ABB RAPID module: ReplayTargets_v20.mod

MODULE ReplayTargets_v20
    ! Generated from tests_v20.csv and success_v20.csv.
    ! Target names include version and testId. B* variants include version, testId, and confId.

    ! Robtargets and jointtargets for replay
    CONST robtarget rA_v20_t1 := [[2348.43,-0.0291239,345.047],[0.199058,0.678508,0.678515,0.199049],[-1,-1,-4,0],[9E+09,9E+09,9E+09,9E+09,9E+09,9E+09]];
    CONST robtarget rB_v20_t1 := [[2448.23,15.5994,307.458],[0.265046,0.716851,0.60792,0.215193],[-1,-1,-4,0],[9E+09,9E+09,9E+09,9E+09,9E+09,9E+09]];
    CONST robtarget rB_v20_t1_c2 := [[2448.23,15.5994,307.458],[0.265046,0.716851,0.60792,0.215193],[0,0,-4,0],[9E+09,9E+09,9E+09,9E+09,9E+09,9E+09]];
    CONST jointtarget jA_v20_t1 := [[-0.000703123,42.2,5.7,-0.000639588,9.4,-270.001],[9E+09,9E+09,9E+09,9E+09,9E+09,9E+09]];
    CONST jointtarget jB_v20_t1 := [[44.9994,-58.7,29.3,-90.0002,39.2,-360.001],[9E+09,9E+09,9E+09,9E+09,9E+09,9E+09]];
    CONST jointtarget jBseed_v20_t1 := [[0,42.2,5.7,0,9.4,-270],[9E+09,9E+09,9E+09,9E+09,9E+09,9E+09]];
    CONST num seedB_v20_t1 := 26880;

    CONST robtarget rA_v20_t2 := [[-1479.72,1306.42,1538.84],[0.318675,0.68714,-0.344424,-0.554668],[1,-4,-1,0],[9E+09,9E+09,9E+09,9E+09,9E+09,9E+09]];
    CONST robtarget rB_v20_t2 := [[-1474.64,1359.47,1499.34],[0.343208,0.716755,-0.240423,-0.557376],[1,-4,-1,0],[9E+09,9E+09,9E+09,9E+09,9E+09,9E+09]];
    CONST robtarget rB_v20_t2_c4 := [[-1474.64,1359.47,1499.34],[0.343208,0.716755,-0.240423,-0.557376],[0,-4,0,0],[9E+09,9E+09,9E+09,9E+09,9E+09,9E+09]];
    CONST jointtarget jA_v20_t2 := [[135,-0.2,15.7,-270,47.2,-45.0005],[9E+09,9E+09,9E+09,9E+09,9E+09,9E+09]];
    CONST jointtarget jB_v20_t2 := [[44.9994,-58.7,29.3,-90.0002,39.2,-360.001],[9E+09,9E+09,9E+09,9E+09,9E+09,9E+09]];
    CONST jointtarget jBseed_v20_t2 := [[135,-0.2,15.7,-270,47.2,-45],[9E+09,9E+09,9E+09,9E+09,9E+09,9E+09]];
    CONST num seedB_v20_t2 := 8986;

    CONST robtarget rA_v20_t3 := [[-971.424,971.394,2079.64],[1.34054E-5,0.567678,-0.567677,-0.596225],[1,0,-4,0],[9E+09,9E+09,9E+09,9E+09,9E+09,9E+09]];
    CONST robtarget rB_v20_t3 := [[-1027.84,1052.99,2102.83],[0.00324872,0.494172,-0.597172,-0.631798],[1,0,-4,0],[9E+09,9E+09,9E+09,9E+09,9E+09,9E+09]];
    CONST robtarget rB_v20_t3_c2 := [[-1027.84,1052.99,2102.83],[0.00324872,0.494172,-0.597172,-0.631798],[0,0,-4,0],[9E+09,9E+09,9E+09,9E+09,9E+09,9E+09]];
    CONST jointtarget jA_v20_t3 := [[135.001,-31.4,20,0.000962912,28.2,-315],[9E+09,9E+09,9E+09,9E+09,9E+09,9E+09]];
    CONST jointtarget jB_v20_t3 := [[44.9994,-58.7,29.3,-90.0002,39.2,-360.001],[9E+09,9E+09,9E+09,9E+09,9E+09,9E+09]];
    CONST jointtarget jBseed_v20_t3 := [[135,-31.4,20,0,28.2,-315],[9E+09,9E+09,9E+09,9E+09,9E+09,9E+09]];
    CONST num seedB_v20_t3 := 10305;

    CONST robtarget rA_v20_t4 := [[-87.9993,-1983.55,1057.37],[0.0429391,-0.444605,-0.7263,0.522466],[-1,2,-4,0],[9E+09,9E+09,9E+09,9E+09,9E+09,9E+09]];
    CONST robtarget rB_v20_t4 := [[-13.7229,-1932.17,1079.47],[0.049502,-0.443461,-0.708683,0.546499],[-1,2,-4,0],[9E+09,9E+09,9E+09,9E+09,9E+09,9E+09]];
    CONST robtarget rB_v20_t4_c3 := [[-13.7229,-1932.17,1079.47],[0.049502,-0.443461,-0.708683,0.546499],[0,4,-4,0],[9E+09,9E+09,9E+09,9E+09,9E+09,9E+09]];
    CONST jointtarget jA_v20_t4 := [[-89.9999,6.4,25.6,270,31.8,-315],[9E+09,9E+09,9E+09,9E+09,9E+09,9E+09]];
    CONST jointtarget jB_v20_t4 := [[44.9994,-58.7,29.3,-90.0002,39.2,-360.001],[9E+09,9E+09,9E+09,9E+09,9E+09,9E+09]];
    CONST jointtarget jBseed_v20_t4 := [[-90,6.4,25.6,270,31.8,-315],[9E+09,9E+09,9E+09,9E+09,9E+09,9E+09]];
    CONST num seedB_v20_t4 := 13879;

    CONST robtarget rA_v20_t5 := [[-1618.75,1500.97,2623.16],[0.821125,-0.204966,-0.515033,0.135956],[1,1,1,0],[9E+09,9E+09,9E+09,9E+09,9E+09,9E+09]];
    CONST robtarget rB_v20_t5 := [[-1548.36,1545.2,2531.64],[0.862384,-0.207508,-0.444636,0.124636],[1,1,1,0],[9E+09,9E+09,9E+09,9E+09,9E+09,9E+09]];
    CONST robtarget rB_v20_t5_c5 := [[-1548.36,1545.2,2531.64],[0.862384,-0.207508,-0.444636,0.124636],[0,0,0,0],[9E+09,9E+09,9E+09,9E+09,9E+09,9E+09]];
    CONST jointtarget jA_v20_t5 := [[135.001,24.2,-50.6,90.0008,29.9,135],[9E+09,9E+09,9E+09,9E+09,9E+09,9E+09]];
    CONST jointtarget jB_v20_t5 := [[44.9994,-58.7,29.3,-90.0002,39.2,-360.001],[9E+09,9E+09,9E+09,9E+09,9E+09,9E+09]];
    CONST jointtarget jBseed_v20_t5 := [[135,24.2,-50.6,90,29.9,135],[9E+09,9E+09,9E+09,9E+09,9E+09,9E+09]];
    CONST num seedB_v20_t5 := 13200;

    CONST robtarget rA_v20_t6 := [[-0.00301178,-325.583,2816.94],[0.976672,0.214735,1.31208E-6,-1.04287E-5],[-2,-3,-2,0],[9E+09,9E+09,9E+09,9E+09,9E+09,9E+09]];
    CONST robtarget rB_v20_t6 := [[12.1082,-256.874,2819],[0.966244,0.241594,-0.061799,0.0646911],[-2,-3,-2,0],[9E+09,9E+09,9E+09,9E+09,9E+09,9E+09]];
    CONST robtarget rB_v20_t6_c4 := [[12.1082,-256.874,2819],[0.966244,0.241594,-0.061799,0.0646911],[0,-4,0,0],[9E+09,9E+09,9E+09,9E+09,9E+09,9E+09]];
    CONST jointtarget jA_v20_t6 := [[-90.0006,-53,2.5,-180.001,14.7,-90.0001],[9E+09,9E+09,9E+09,9E+09,9E+09,9E+09]];
    CONST jointtarget jB_v20_t6 := [[44.9994,-58.7,29.3,-90.0002,39.2,-360.001],[9E+09,9E+09,9E+09,9E+09,9E+09,9E+09]];
    CONST jointtarget jBseed_v20_t6 := [[-90,-53,2.5,-180,14.7,-90],[9E+09,9E+09,9E+09,9E+09,9E+09,9E+09]];
    CONST num seedB_v20_t6 := 26677;

    CONST robtarget rA_v20_t7 := [[1448.08,-93.8143,1159.42],[0.151545,0.78397,-0.512149,0.316431],[-1,-1,-2,0],[9E+09,9E+09,9E+09,9E+09,9E+09,9E+09]];
    CONST robtarget rB_v20_t7 := [[1454.33,-138.013,1185.15],[0.132933,0.822904,-0.460863,0.304569],[-1,-1,-2,0],[9E+09,9E+09,9E+09,9E+09,9E+09,9E+09]];
    CONST robtarget rB_v20_t7_c5 := [[1454.33,-138.013,1185.15],[0.132933,0.822904,-0.460863,0.304569],[0,0,0,0],[9E+09,9E+09,9E+09,9E+09,9E+09,9E+09]];
    CONST robtarget rB_v20_t7_c8 := [[1454.33,-138.013,1185.15],[0.132933,0.822904,-0.460863,0.304569],[0,0,4,0],[9E+09,9E+09,9E+09,9E+09,9E+09,9E+09]];
    CONST jointtarget jA_v20_t7 := [[-0.000199191,-22.7,45.6,-44.9996,52.6,-90.0001],[9E+09,9E+09,9E+09,9E+09,9E+09,9E+09]];
    CONST jointtarget jB_v20_t7 := [[44.9994,-58.7,29.3,-90.0002,39.2,-360.001],[9E+09,9E+09,9E+09,9E+09,9E+09,9E+09]];
    CONST jointtarget jBseed_v20_t7 := [[0,-22.7,45.6,-45,52.6,-90],[9E+09,9E+09,9E+09,9E+09,9E+09,9E+09]];
    CONST num seedB_v20_t7 := 27772;

    CONST robtarget rA_v20_t8 := [[1676.32,-1692.34,1208.08],[0.539776,0.76394,0.296429,0.192788],[-1,2,2,0],[9E+09,9E+09,9E+09,9E+09,9E+09,9E+09]];
    CONST robtarget rB_v20_t8 := [[1594.8,-1750.16,1141.03],[0.532215,0.796727,0.236675,0.161115],[-1,2,2,0],[9E+09,9E+09,9E+09,9E+09,9E+09,9E+09]];
    CONST robtarget rB_v20_t8_c5 := [[1594.8,-1750.16,1141.03],[0.532215,0.796727,0.236675,0.161115],[0,0,0,0],[9E+09,9E+09,9E+09,9E+09,9E+09,9E+09]];
    CONST robtarget rB_v20_t8_c6 := [[1594.8,-1750.16,1141.03],[0.532215,0.796727,0.236675,0.161115],[0,4,0,0],[9E+09,9E+09,9E+09,9E+09,9E+09,9E+09]];
    CONST jointtarget jA_v20_t8 := [[-45.0002,21.5,2.5,225,5.5,225.001],[9E+09,9E+09,9E+09,9E+09,9E+09,9E+09]];
    CONST jointtarget jB_v20_t8 := [[44.9994,-58.7,29.3,-90.0002,39.2,-360.001],[9E+09,9E+09,9E+09,9E+09,9E+09,9E+09]];
    CONST jointtarget jBseed_v20_t8 := [[-45,21.5,2.5,225,5.5,225],[9E+09,9E+09,9E+09,9E+09,9E+09,9E+09]];
    CONST num seedB_v20_t8 := 3525;

    CONST robtarget rA_v20_t9 := [[-1079.34,1079.34,1641.75],[0.71135,-0.589521,-0.244195,0.294643],[1,1,0,0],[9E+09,9E+09,9E+09,9E+09,9E+09,9E+09]];
    CONST robtarget rB_v20_t9 := [[-966.677,1102.66,1605.56],[0.710962,-0.602204,-0.160651,0.325692],[1,1,0,0],[9E+09,9E+09,9E+09,9E+09,9E+09,9E+09]];
    CONST robtarget rB_v20_t9_c4 := [[-966.677,1102.66,1605.56],[0.710962,-0.602204,-0.160651,0.325692],[0,-4,0,0],[9E+09,9E+09,9E+09,9E+09,9E+09,9E+09]];
    CONST robtarget rB_v20_t9_c5 := [[-966.677,1102.66,1605.56],[0.710962,-0.602204,-0.160651,0.325692],[0,0,0,0],[9E+09,9E+09,9E+09,9E+09,9E+09,9E+09]];
    CONST jointtarget jA_v20_t9 := [[135,-27.5,36.8,179.999,20,89.9998],[9E+09,9E+09,9E+09,9E+09,9E+09,9E+09]];
    CONST jointtarget jB_v20_t9 := [[44.9994,-58.7,29.3,-90.0002,39.2,-360.001],[9E+09,9E+09,9E+09,9E+09,9E+09,9E+09]];
    CONST jointtarget jBseed_v20_t9 := [[135,-27.5,36.8,180,20,90],[9E+09,9E+09,9E+09,9E+09,9E+09,9E+09]];
    CONST num seedB_v20_t9 := 19894;

    CONST robtarget rA_v20_t10 := [[138.442,2028.98,2186.31],[0.730348,-0.405331,0.548774,-0.0338534],[1,-1,-4,0],[9E+09,9E+09,9E+09,9E+09,9E+09,9E+09]];
    CONST robtarget rB_v20_t10 := [[136.362,1909.01,2210.89],[0.67858,-0.463529,0.560222,-0.104029],[1,-1,-4,0],[9E+09,9E+09,9E+09,9E+09,9E+09,9E+09]];
    CONST robtarget rB_v20_t10_c2 := [[136.362,1909.01,2210.89],[0.67858,-0.463529,0.560222,-0.104029],[0,0,-4,0],[9E+09,9E+09,9E+09,9E+09,9E+09,9E+09]];
    CONST jointtarget jA_v20_t10 := [[90.0002,5.4,-12.5,-89.9994,56,-315],[9E+09,9E+09,9E+09,9E+09,9E+09,9E+09]];
    CONST jointtarget jB_v20_t10 := [[44.9994,-58.7,29.3,-90.0002,39.2,-360.001],[9E+09,9E+09,9E+09,9E+09,9E+09,9E+09]];
    CONST jointtarget jBseed_v20_t10 := [[90,5.4,-12.5,-90,56,-315],[9E+09,9E+09,9E+09,9E+09,9E+09,9E+09]];
    CONST num seedB_v20_t10 := 2946;

    CONST robtarget rA_v20_t11 := [[1156.13,1172.74,2229.26],[0.716045,-0.261719,0.561783,0.321221],[0,1,2,0],[9E+09,9E+09,9E+09,9E+09,9E+09,9E+09]];
    CONST robtarget rB_v20_t11 := [[1235.48,1131.05,2183.34],[0.723682,-0.214068,0.602425,0.259892],[0,1,2,0],[9E+09,9E+09,9E+09,9E+09,9E+09,9E+09]];
    CONST robtarget rB_v20_t11_c6 := [[1235.48,1131.05,2183.34],[0.723682,-0.214068,0.602425,0.259892],[0,4,0,0],[9E+09,9E+09,9E+09,9E+09,9E+09,9E+09]];
    CONST jointtarget jA_v20_t11 := [[45.0005,-17.1,7.7,135,5.7,225.001],[9E+09,9E+09,9E+09,9E+09,9E+09,9E+09]];
    CONST jointtarget jB_v20_t11 := [[44.9994,-58.7,29.3,-90.0002,39.2,-360.001],[9E+09,9E+09,9E+09,9E+09,9E+09,9E+09]];
    CONST jointtarget jBseed_v20_t11 := [[45,-17.1,7.7,135,5.7,225],[9E+09,9E+09,9E+09,9E+09,9E+09,9E+09]];
    CONST num seedB_v20_t11 := 2997;

    CONST robtarget rA_v20_t12 := [[2684.36,-73.5564,2199.23],[0.910091,0.192131,0.342612,-0.132052],[-1,-2,1,0],[9E+09,9E+09,9E+09,9E+09,9E+09,9E+09]];
    CONST robtarget rB_v20_t12 := [[2614.98,29.0324,2213.55],[0.904293,0.217033,0.287629,-0.228955],[-1,-2,1,0],[9E+09,9E+09,9E+09,9E+09,9E+09,9E+09]];
    CONST robtarget rB_v20_t12_c4 := [[2614.98,29.0324,2213.55],[0.904293,0.217033,0.287629,-0.228955],[0,-4,0,0],[9E+09,9E+09,9E+09,9E+09,9E+09,9E+09]];
    CONST jointtarget jA_v20_t12 := [[-0.000960234,53.1,-74.1,-135,38.5,135],[9E+09,9E+09,9E+09,9E+09,9E+09,9E+09]];
    CONST jointtarget jB_v20_t12 := [[44.9994,-58.7,29.3,-90.0002,39.2,-360.001],[9E+09,9E+09,9E+09,9E+09,9E+09,9E+09]];
    CONST jointtarget jBseed_v20_t12 := [[0,53.1,-74.1,-135,38.5,135],[9E+09,9E+09,9E+09,9E+09,9E+09,9E+09]];
    CONST num seedB_v20_t12 := 170;

    CONST robtarget rA_v20_t13 := [[0.00419857,298.28,3136.24],[0.368757,-0.102269,-0.246896,-0.890282],[0,-1,-3,0],[9E+09,9E+09,9E+09,9E+09,9E+09,9E+09]];
    CONST robtarget rB_v20_t13 := [[-28.1699,255.485,3048.95],[0.422465,-0.149707,-0.227149,-0.864589],[0,-1,-3,0],[9E+09,9E+09,9E+09,9E+09,9E+09,9E+09]];
    CONST robtarget rB_v20_t13_c5 := [[-28.1699,255.485,3048.95],[0.422465,-0.149707,-0.227149,-0.864589],[0,0,0,0],[9E+09,9E+09,9E+09,9E+09,9E+09,9E+09]];
    CONST jointtarget jA_v20_t13 := [[89.9992,-38.4,-22.1,-0.000207024,1.5,-225],[9E+09,9E+09,9E+09,9E+09,9E+09,9E+09]];
    CONST jointtarget jB_v20_t13 := [[44.9994,-58.7,29.3,-90.0002,39.2,-360.001],[9E+09,9E+09,9E+09,9E+09,9E+09,9E+09]];
    CONST jointtarget jBseed_v20_t13 := [[90,-38.4,-22.1,0,1.5,-225],[9E+09,9E+09,9E+09,9E+09,9E+09,9E+09]];
    CONST num seedB_v20_t13 := 21910;

    CONST robtarget rA_v20_t14 := [[-217.284,360.724,3378.8],[0.700643,0.169716,0.342315,0.602592],[1,2,-3,0],[9E+09,9E+09,9E+09,9E+09,9E+09,9E+09]];
    CONST robtarget rB_v20_t14 := [[-203.6,421.862,3270.5],[0.694668,0.134709,0.317582,0.631214],[1,2,-3,0],[9E+09,9E+09,9E+09,9E+09,9E+09,9E+09]];
    CONST robtarget rB_v20_t14_c3 := [[-203.6,421.862,3270.5],[0.694668,0.134709,0.317582,0.631214],[0,4,-4,0],[9E+09,9E+09,9E+09,9E+09,9E+09,9E+09]];
    CONST jointtarget jA_v20_t14 := [[135,-13.9,-53.2,224.999,59.2,-269.999],[9E+09,9E+09,9E+09,9E+09,9E+09,9E+09]];
    CONST jointtarget jB_v20_t14 := [[44.9994,-58.7,29.3,-90.0002,39.2,-360.001],[9E+09,9E+09,9E+09,9E+09,9E+09,9E+09]];
    CONST jointtarget jBseed_v20_t14 := [[135,-13.9,-53.2,225,59.2,-270],[9E+09,9E+09,9E+09,9E+09,9E+09,9E+09]];
    CONST num seedB_v20_t14 := 4792;

    CONST robtarget rA_v20_t15 := [[-1472.6,1608.71,1063.4],[0.00433901,0.101786,-0.642952,-0.7591],[1,2,2,0],[9E+09,9E+09,9E+09,9E+09,9E+09,9E+09]];
    CONST robtarget rB_v20_t15 := [[-1457.34,1584.84,1032.33],[0.104698,-0.085445,0.659952,0.739054],[1,2,2,0],[9E+09,9E+09,9E+09,9E+09,9E+09,9E+09]];
    CONST robtarget rB_v20_t15_c6 := [[-1457.34,1584.84,1032.33],[0.104698,-0.085445,0.659952,0.739054],[0,4,0,0],[9E+09,9E+09,9E+09,9E+09,9E+09,9E+09]];
    CONST jointtarget jA_v20_t15 := [[135,17.2,16.9,225.001,54.6,224.999],[9E+09,9E+09,9E+09,9E+09,9E+09,9E+09]];
    CONST jointtarget jB_v20_t15 := [[44.9994,-58.7,29.3,-90.0002,39.2,-360.001],[9E+09,9E+09,9E+09,9E+09,9E+09,9E+09]];
    CONST jointtarget jBseed_v20_t15 := [[135,17.2,16.9,225,54.6,225],[9E+09,9E+09,9E+09,9E+09,9E+09,9E+09]];
    CONST num seedB_v20_t15 := 4784;

    CONST robtarget rA_v20_t17 := [[-0.0178469,-1454.99,2120.23],[0.807655,0.448611,-0.185819,0.334533],[-2,-3,3,0],[9E+09,9E+09,9E+09,9E+09,9E+09,9E+09]];
    CONST robtarget rB_v20_t17 := [[95.0666,-1392.8,2093],[0.815027,0.420993,-0.246161,0.312891],[-2,-3,3,0],[9E+09,9E+09,9E+09,9E+09,9E+09,9E+09]];
    CONST robtarget rB_v20_t17_c7 := [[95.0666,-1392.8,2093],[0.815027,0.420993,-0.246161,0.312891],[0,-4,4,0],[9E+09,9E+09,9E+09,9E+09,9E+09,9E+09]];
    CONST jointtarget jA_v20_t17 := [[-90.0007,-27.8,21.4,-180.001,25.5,315],[9E+09,9E+09,9E+09,9E+09,9E+09,9E+09]];
    CONST jointtarget jB_v20_t17 := [[44.9994,-58.7,29.3,-90.0002,39.2,-360.001],[9E+09,9E+09,9E+09,9E+09,9E+09,9E+09]];
    CONST jointtarget jBseed_v20_t17 := [[-90,-27.8,21.4,-180,25.5,315],[9E+09,9E+09,9E+09,9E+09,9E+09,9E+09]];
    CONST num seedB_v20_t17 := 20361;

    CONST robtarget rA_v20_t19 := [[-0.0210649,1955.73,510.213],[0.382393,-0.841027,-0.348368,-0.158391],[1,2,0,0],[9E+09,9E+09,9E+09,9E+09,9E+09,9E+09]];
    CONST robtarget rB_v20_t19 := [[49.9779,1894.06,474.945],[0.404386,-0.810845,-0.415016,-0.0822396],[1,2,0,0],[9E+09,9E+09,9E+09,9E+09,9E+09,9E+09]];
    CONST robtarget rB_v20_t19_c5 := [[49.9779,1894.06,474.945],[0.404386,-0.810845,-0.415016,-0.0822396],[0,0,0,0],[9E+09,9E+09,9E+09,9E+09,9E+09,9E+09]];
    CONST jointtarget jA_v20_t19 := [[90.0006,20.9,31.1,180.001,10.9,44.9993],[9E+09,9E+09,9E+09,9E+09,9E+09,9E+09]];
    CONST jointtarget jB_v20_t19 := [[44.9994,-58.7,29.3,-90.0002,39.2,-360.001],[9E+09,9E+09,9E+09,9E+09,9E+09,9E+09]];
    CONST jointtarget jBseed_v20_t19 := [[90,20.9,31.1,180,10.9,45],[9E+09,9E+09,9E+09,9E+09,9E+09,9E+09]];
    CONST num seedB_v20_t19 := 31692;

    CONST robtarget rA_v20_t20 := [[238.468,195.527,2977.81],[0.329804,-0.375038,-0.0601945,-0.864264],[0,-1,-2,0],[9E+09,9E+09,9E+09,9E+09,9E+09,9E+09]];
    CONST robtarget rB_v20_t20 := [[269.534,283.158,2926.07],[0.244024,-0.333193,0.0131063,-0.910639],[0,-1,-2,0],[9E+09,9E+09,9E+09,9E+09,9E+09,9E+09]];
    CONST robtarget rB_v20_t20_c5 := [[269.534,283.158,2926.07],[0.244024,-0.333193,0.0131063,-0.910639],[0,0,0,0],[9E+09,9E+09,9E+09,9E+09,9E+09,9E+09]];
    CONST robtarget rB_v20_t20_c6 := [[269.534,283.158,2926.07],[0.244024,-0.333193,0.0131063,-0.910639],[0,4,0,0],[9E+09,9E+09,9E+09,9E+09,9E+09,9E+09]];
    CONST jointtarget jA_v20_t20 := [[45.0001,-45.7,-11.3,-45.0005,14.9,-135],[9E+09,9E+09,9E+09,9E+09,9E+09,9E+09]];
    CONST jointtarget jB_v20_t20 := [[44.9994,-58.7,29.3,-90.0002,39.2,-360.001],[9E+09,9E+09,9E+09,9E+09,9E+09,9E+09]];
    CONST jointtarget jBseed_v20_t20 := [[45,-45.7,-11.3,-45,14.9,-135],[9E+09,9E+09,9E+09,9E+09,9E+09,9E+09]];
    CONST num seedB_v20_t20 := 23746;

    CONST robtarget rA_v20_t22 := [[-1109.18,1224.53,1567.08],[0.48889,-0.472376,0.368672,0.633978],[1,-2,-3,0],[9E+09,9E+09,9E+09,9E+09,9E+09,9E+09]];
    CONST robtarget rB_v20_t22 := [[-1201.74,1194.66,1668.32],[0.482702,-0.408187,0.43208,0.643187],[1,-2,-3,0],[9E+09,9E+09,9E+09,9E+09,9E+09,9E+09]];
    CONST robtarget rB_v20_t22_c2 := [[-1201.74,1194.66,1668.32],[0.482702,-0.408187,0.43208,0.643187],[0,0,-4,0],[9E+09,9E+09,9E+09,9E+09,9E+09,9E+09]];
    CONST jointtarget jA_v20_t22 := [[135.001,-18.4,33.6,-135,43.7,-225],[9E+09,9E+09,9E+09,9E+09,9E+09,9E+09]];
    CONST jointtarget jB_v20_t22 := [[44.9994,-58.7,29.3,-90.0002,39.2,-360.001],[9E+09,9E+09,9E+09,9E+09,9E+09,9E+09]];
    CONST jointtarget jBseed_v20_t22 := [[135,-18.4,33.6,-135,43.7,-225],[9E+09,9E+09,9E+09,9E+09,9E+09,9E+09]];
    CONST num seedB_v20_t22 := 27671;

    CONST robtarget rA_v20_t23 := [[1206.08,1190.09,1007.16],[0.219968,0.345403,0.79192,0.45296],[0,2,2,0],[9E+09,9E+09,9E+09,9E+09,9E+09,9E+09]];
    CONST robtarget rB_v20_t23 := [[1249.95,1205.88,924.826],[0.202523,0.303121,0.775905,0.514852],[0,2,2,0],[9E+09,9E+09,9E+09,9E+09,9E+09,9E+09]];
    CONST robtarget rB_v20_t23_c8 := [[1249.95,1205.88,924.826],[0.202523,0.303121,0.775905,0.514852],[0,0,4,0],[9E+09,9E+09,9E+09,9E+09,9E+09,9E+09]];
    CONST jointtarget jA_v20_t23 := [[45.0003,-8.8,42.3,225.001,5.5,224.999],[9E+09,9E+09,9E+09,9E+09,9E+09,9E+09]];
    CONST jointtarget jB_v20_t23 := [[44.9994,-58.7,29.3,-90.0002,39.2,-360.001],[9E+09,9E+09,9E+09,9E+09,9E+09,9E+09]];
    CONST jointtarget jBseed_v20_t23 := [[45,-8.8,42.3,225,5.5,225],[9E+09,9E+09,9E+09,9E+09,9E+09,9E+09]];
    CONST num seedB_v20_t23 := 137;

    CONST robtarget rA_v20_t24 := [[97.7592,-1489.52,-79.8919],[0.163535,-0.345966,0.795226,-0.470296],[-2,1,-4,0],[9E+09,9E+09,9E+09,9E+09,9E+09,9E+09]];
    CONST robtarget rB_v20_t24 := [[103.375,-1616.07,-25.6002],[0.193183,-0.292041,0.785636,-0.510068],[-2,1,-4,0],[9E+09,9E+09,9E+09,9E+09,9E+09,9E+09]];
    CONST robtarget rB_v20_t24_c2 := [[103.375,-1616.07,-25.6002],[0.193183,-0.292041,0.785636,-0.510068],[0,0,-4,0],[9E+09,9E+09,9E+09,9E+09,9E+09,9E+09]];
    CONST jointtarget jA_v20_t24 := [[-90.0009,40.1,44.6,135.001,55.9,-270],[9E+09,9E+09,9E+09,9E+09,9E+09,9E+09]];
    CONST jointtarget jB_v20_t24 := [[44.9994,-58.7,29.3,-90.0002,39.2,-360.001],[9E+09,9E+09,9E+09,9E+09,9E+09,9E+09]];
    CONST jointtarget jBseed_v20_t24 := [[-90,40.1,44.6,135,55.9,-270],[9E+09,9E+09,9E+09,9E+09,9E+09,9E+09]];
    CONST num seedB_v20_t24 := 32351;

    CONST robtarget rA_v20_t25 := [[125.84,-2076.87,2190.37],[0.273438,-0.310714,0.60141,-0.68337],[-2,-4,1,0],[9E+09,9E+09,9E+09,9E+09,9E+09,9E+09]];
    CONST robtarget rB_v20_t25 := [[220.204,-2033.24,2142.64],[0.243299,-0.295957,0.561806,-0.733204],[-2,-4,1,0],[9E+09,9E+09,9E+09,9E+09,9E+09,9E+09]];
    CONST robtarget rB_v20_t25_c4 := [[220.204,-2033.24,2142.64],[0.243299,-0.295957,0.561806,-0.733204],[0,-4,0,0],[9E+09,9E+09,9E+09,9E+09,9E+09,9E+09]];
    CONST jointtarget jA_v20_t25 := [[-90.0001,7.1,-14.4,-270,48.9,179.999],[9E+09,9E+09,9E+09,9E+09,9E+09,9E+09]];
    CONST jointtarget jB_v20_t25 := [[44.9994,-58.7,29.3,-90.0002,39.2,-360.001],[9E+09,9E+09,9E+09,9E+09,9E+09,9E+09]];
    CONST jointtarget jBseed_v20_t25 := [[-90,7.1,-14.4,-270,48.9,180],[9E+09,9E+09,9E+09,9E+09,9E+09,9E+09]];
    CONST num seedB_v20_t25 := 30175;

    CONST robtarget rA_v20_t27 := [[1918.58,-2031.81,1938.35],[0.0914884,-0.0961396,0.777017,-0.615331],[-1,-1,-1,0],[9E+09,9E+09,9E+09,9E+09,9E+09,9E+09]];
    CONST robtarget rB_v20_t27 := [[1897.77,-2061.28,1842.5],[0.000557429,0.128274,-0.779554,0.613058],[-1,-1,-1,0],[9E+09,9E+09,9E+09,9E+09,9E+09,9E+09]];
    CONST robtarget rB_v20_t27_c5 := [[1897.77,-2061.28,1842.5],[0.000557429,0.128274,-0.779554,0.613058],[0,0,0,0],[9E+09,9E+09,9E+09,9E+09,9E+09,9E+09]];
    CONST jointtarget jA_v20_t27 := [[-44.9997,55.6,-73.8,-45.0007,42.7,-44.9995],[9E+09,9E+09,9E+09,9E+09,9E+09,9E+09]];
    CONST jointtarget jB_v20_t27 := [[44.9994,-58.7,29.3,-90.0002,39.2,-360.001],[9E+09,9E+09,9E+09,9E+09,9E+09,9E+09]];
    CONST jointtarget jBseed_v20_t27 := [[-45,55.6,-73.8,-45,42.7,-45],[9E+09,9E+09,9E+09,9E+09,9E+09,9E+09]];
    CONST num seedB_v20_t27 := 30351;

    CONST robtarget rA_v20_t28 := [[13.7981,2914.82,1743.86],[0.779438,-0.625115,0.0311377,-0.0271682],[0,-2,0,0],[9E+09,9E+09,9E+09,9E+09,9E+09,9E+09]];
    CONST robtarget rB_v20_t28 := [[13.1914,2858.61,1667.39],[0.807694,-0.57037,0.0537412,-0.139357],[0,-2,0,0],[9E+09,9E+09,9E+09,9E+09,9E+09,9E+09]];
    CONST robtarget rB_v20_t28_c4 := [[13.1914,2858.61,1667.39],[0.807694,-0.57037,0.0537412,-0.139357],[0,-4,0,0],[9E+09,9E+09,9E+09,9E+09,9E+09,9E+09]];
    CONST jointtarget jA_v20_t28 := [[89.9996,55.8,-63.6,-134.999,6.7,44.9991],[9E+09,9E+09,9E+09,9E+09,9E+09,9E+09]];
    CONST jointtarget jB_v20_t28 := [[44.9994,-58.7,29.3,-90.0002,39.2,-360.001],[9E+09,9E+09,9E+09,9E+09,9E+09,9E+09]];
    CONST jointtarget jBseed_v20_t28 := [[90,55.8,-63.6,-135,6.7,45],[9E+09,9E+09,9E+09,9E+09,9E+09,9E+09]];
    CONST num seedB_v20_t28 := 16775;

    CONST robtarget rA_v20_t29 := [[-1462.15,-1378.18,-139.572],[0.181517,-0.672723,-0.628398,0.345849],[-2,-2,-4,0],[9E+09,9E+09,9E+09,9E+09,9E+09,9E+09]];
    CONST robtarget rB_v20_t29 := [[-1363.66,-1277.19,-121.909],[0.186146,-0.700461,-0.59665,0.344547],[-2,-2,-4,0],[9E+09,9E+09,9E+09,9E+09,9E+09,9E+09]];
    CONST robtarget rB_v20_t29_c2 := [[-1363.66,-1277.19,-121.909],[0.186146,-0.700461,-0.59665,0.344547],[0,0,-4,0],[9E+09,9E+09,9E+09,9E+09,9E+09,9E+09]];
    CONST jointtarget jA_v20_t29 := [[-134.999,51.5,18.9,-135,30.2,-270.001],[9E+09,9E+09,9E+09,9E+09,9E+09,9E+09]];
    CONST jointtarget jB_v20_t29 := [[44.9994,-58.7,29.3,-90.0002,39.2,-360.001],[9E+09,9E+09,9E+09,9E+09,9E+09,9E+09]];
    CONST jointtarget jBseed_v20_t29 := [[-135,51.5,18.9,-135,30.2,-270],[9E+09,9E+09,9E+09,9E+09,9E+09,9E+09]];
    CONST num seedB_v20_t29 := 9727;

    CONST robtarget rA_v20_t30 := [[375.616,421.367,3490.03],[0.6792,-0.0971219,0.213528,0.695457],[0,0,-1,0],[9E+09,9E+09,9E+09,9E+09,9E+09,9E+09]];
    CONST robtarget rB_v20_t30 := [[393.212,359.456,3471.37],[0.700033,-0.120448,0.296069,0.638584],[0,0,-1,0],[9E+09,9E+09,9E+09,9E+09,9E+09,9E+09]];
    CONST robtarget rB_v20_t30_c5 := [[393.212,359.456,3471.37],[0.700033,-0.120448,0.296069,0.638584],[0,0,0,0],[9E+09,9E+09,9E+09,9E+09,9E+09,9E+09]];
    CONST jointtarget jA_v20_t30 := [[44.9999,0.4,-76.9,45.0006,15.9,-0.000480438],[9E+09,9E+09,9E+09,9E+09,9E+09,9E+09]];
    CONST jointtarget jB_v20_t30 := [[44.9994,-58.7,29.3,-90.0002,39.2,-360.001],[9E+09,9E+09,9E+09,9E+09,9E+09,9E+09]];
    CONST jointtarget jBseed_v20_t30 := [[45,0.4,-76.9,45,15.9,0],[9E+09,9E+09,9E+09,9E+09,9E+09,9E+09]];
    CONST num seedB_v20_t30 := 31577;

    CONST robtarget rA_v20_t31 := [[2378.29,-10.2339,1148.77],[0.180245,-0.774747,0.338557,-0.502651],[-1,-1,-1,0],[9E+09,9E+09,9E+09,9E+09,9E+09,9E+09]];
    CONST robtarget rB_v20_t31 := [[2418.67,18.3615,1021.64],[0.188844,-0.810787,0.272248,-0.482539],[-1,-1,-1,0],[9E+09,9E+09,9E+09,9E+09,9E+09,9E+09]];
    CONST robtarget rB_v20_t31_c4 := [[2418.67,18.3615,1021.64],[0.188844,-0.810787,0.272248,-0.482539],[0,-4,0,0],[9E+09,9E+09,9E+09,9E+09,9E+09,9E+09]];
    CONST robtarget rB_v20_t31_c5 := [[2418.67,18.3615,1021.64],[0.188844,-0.810787,0.272248,-0.482539],[0,0,0,0],[9E+09,9E+09,9E+09,9E+09,9E+09,9E+09]];
    CONST jointtarget jA_v20_t31 := [[-0.000935507,22.3,3.2,-89.9999,3.5,-45],[9E+09,9E+09,9E+09,9E+09,9E+09,9E+09]];
    CONST jointtarget jB_v20_t31 := [[44.9994,-58.7,29.3,-90.0002,39.2,-360.001],[9E+09,9E+09,9E+09,9E+09,9E+09,9E+09]];
    CONST jointtarget jBseed_v20_t31 := [[0,22.3,3.2,-90,3.5,-45],[9E+09,9E+09,9E+09,9E+09,9E+09,9E+09]];
    CONST num seedB_v20_t31 := 15059;

    CONST robtarget rA_v20_t32 := [[-1677.05,1857.4,162.463],[0.242382,-0.188474,0.841235,0.445031],[1,-1,-2,0],[9E+09,9E+09,9E+09,9E+09,9E+09,9E+09]];
    CONST robtarget rB_v20_t32 := [[-1685.95,1794.1,90.0996],[0.175293,-0.159407,0.873711,0.424841],[1,-1,-2,0],[9E+09,9E+09,9E+09,9E+09,9E+09,9E+09]];
    CONST robtarget rB_v20_t32_c2 := [[-1685.95,1794.1,90.0996],[0.175293,-0.159407,0.873711,0.424841],[0,0,-4,0],[9E+09,9E+09,9E+09,9E+09,9E+09,9E+09]];
    CONST jointtarget jA_v20_t32 := [[135.001,57.1,-8.2,-89.9996,49.8,-179.999],[9E+09,9E+09,9E+09,9E+09,9E+09,9E+09]];
    CONST jointtarget jB_v20_t32 := [[44.9994,-58.7,29.3,-90.0002,39.2,-360.001],[9E+09,9E+09,9E+09,9E+09,9E+09,9E+09]];
    CONST jointtarget jBseed_v20_t32 := [[135,57.1,-8.2,-90,49.8,-180],[9E+09,9E+09,9E+09,9E+09,9E+09,9E+09]];
    CONST num seedB_v20_t32 := 25561;

    CONST robtarget rA_v20_t33 := [[-1713.62,-1775.86,696.337],[0.458173,0.370152,-0.741708,0.320832],[-2,1,0,0],[9E+09,9E+09,9E+09,9E+09,9E+09,9E+09]];
    CONST robtarget rB_v20_t33 := [[-1721.55,-1822.95,635.019],[0.506835,0.31009,-0.735215,0.326223],[-2,1,0,0],[9E+09,9E+09,9E+09,9E+09,9E+09,9E+09]];
    CONST robtarget rB_v20_t33_c4 := [[-1721.55,-1822.95,635.019],[0.506835,0.31009,-0.735215,0.326223],[0,-4,0,0],[9E+09,9E+09,9E+09,9E+09,9E+09,9E+09]];
    CONST robtarget rB_v20_t33_c5 := [[-1721.55,-1822.95,635.019],[0.506835,0.31009,-0.735215,0.326223],[0,0,0,0],[9E+09,9E+09,9E+09,9E+09,9E+09,9E+09]];
    CONST jointtarget jA_v20_t33 := [[-135.001,36.5,2.2,135.001,21.9,44.9992],[9E+09,9E+09,9E+09,9E+09,9E+09,9E+09]];
    CONST jointtarget jB_v20_t33 := [[44.9994,-58.7,29.3,-90.0002,39.2,-360.001],[9E+09,9E+09,9E+09,9E+09,9E+09,9E+09]];
    CONST jointtarget jBseed_v20_t33 := [[-135,36.5,2.2,135,21.9,45],[9E+09,9E+09,9E+09,9E+09,9E+09,9E+09]];
    CONST num seedB_v20_t33 := 28196;

    CONST robtarget rA_v20_t34 := [[-839.919,839.899,2858.77],[0.240829,-0.71799,0.2974,0.581417],[1,-1,-4,0],[9E+09,9E+09,9E+09,9E+09,9E+09,9E+09]];
    CONST robtarget rB_v20_t34 := [[-766.287,889.177,2826.58],[0.185995,-0.714842,0.355007,0.573041],[1,-1,-4,0],[9E+09,9E+09,9E+09,9E+09,9E+09,9E+09]];
    CONST robtarget rB_v20_t34_c2 := [[-766.287,889.177,2826.58],[0.185995,-0.714842,0.355007,0.573041],[0,0,-4,0],[9E+09,9E+09,9E+09,9E+09,9E+09,9E+09]];
    CONST jointtarget jA_v20_t34 := [[135.001,-17.8,-22.7,-0.000681613,52.5,-359.999],[9E+09,9E+09,9E+09,9E+09,9E+09,9E+09]];
    CONST jointtarget jB_v20_t34 := [[44.9994,-58.7,29.3,-90.0002,39.2,-360.001],[9E+09,9E+09,9E+09,9E+09,9E+09,9E+09]];
    CONST jointtarget jBseed_v20_t34 := [[135,-17.8,-22.7,0,52.5,-360],[9E+09,9E+09,9E+09,9E+09,9E+09,9E+09]];
    CONST num seedB_v20_t34 := 31998;

    CONST robtarget rA_v20_t35 := [[1351.09,-1449.45,-304.38],[0.399922,0.855014,0.322793,-0.0694059],[-1,-2,-2,0],[9E+09,9E+09,9E+09,9E+09,9E+09,9E+09]];
    CONST robtarget rB_v20_t35 := [[1386.13,-1550.01,-285.387],[0.489421,0.824111,0.277103,-0.0672532],[-1,-2,-2,0],[9E+09,9E+09,9E+09,9E+09,9E+09,9E+09]];
    CONST robtarget rB_v20_t35_c4 := [[1386.13,-1550.01,-285.387],[0.489421,0.824111,0.277103,-0.0672532],[0,-4,0,0],[9E+09,9E+09,9E+09,9E+09,9E+09,9E+09]];
    CONST jointtarget jA_v20_t35 := [[-44.9992,58.9,15.9,-135,36.1,-134.999],[9E+09,9E+09,9E+09,9E+09,9E+09,9E+09]];
    CONST jointtarget jB_v20_t35 := [[44.9994,-58.7,29.3,-90.0002,39.2,-360.001],[9E+09,9E+09,9E+09,9E+09,9E+09,9E+09]];
    CONST jointtarget jBseed_v20_t35 := [[-45,58.9,15.9,-135,36.1,-135],[9E+09,9E+09,9E+09,9E+09,9E+09,9E+09]];
    CONST num seedB_v20_t35 := 1029;

    CONST robtarget rA_v20_t36 := [[76.08,-1964.14,2256.72],[0.479124,0.00265306,0.479385,-0.73527],[-1,-3,2,0],[9E+09,9E+09,9E+09,9E+09,9E+09,9E+09]];
    CONST robtarget rB_v20_t36 := [[76.552,-1875.91,2195.82],[0.448379,0.0363468,0.563891,-0.692576],[-1,-3,2,0],[9E+09,9E+09,9E+09,9E+09,9E+09,9E+09]];
    CONST robtarget rB_v20_t36_c4 := [[76.552,-1875.91,2195.82],[0.448379,0.0363468,0.563891,-0.692576],[0,-4,0,0],[9E+09,9E+09,9E+09,9E+09,9E+09,9E+09]];
    CONST jointtarget jA_v20_t36 := [[-89.9995,0.6,-7.2,-225,40.1,180.001],[9E+09,9E+09,9E+09,9E+09,9E+09,9E+09]];
    CONST jointtarget jB_v20_t36 := [[44.9994,-58.7,29.3,-90.0002,39.2,-360.001],[9E+09,9E+09,9E+09,9E+09,9E+09,9E+09]];
    CONST jointtarget jBseed_v20_t36 := [[-90,0.6,-7.2,-225,40.1,180],[9E+09,9E+09,9E+09,9E+09,9E+09,9E+09]];
    CONST num seedB_v20_t36 := 21562;

    CONST robtarget rA_v20_t37 := [[23.8193,273.657,2922.22],[0.688568,-0.160869,0.257432,0.658577],[0,3,0,0],[9E+09,9E+09,9E+09,9E+09,9E+09,9E+09]];
    CONST robtarget rB_v20_t37 := [[-43.0516,310.601,2870.45],[0.733212,-0.135064,0.216285,0.63038],[0,3,0,0],[9E+09,9E+09,9E+09,9E+09,9E+09,9E+09]];
    CONST robtarget rB_v20_t37_c6 := [[-43.0516,310.601,2870.45],[0.733212,-0.135064,0.216285,0.63038],[0,4,0,0],[9E+09,9E+09,9E+09,9E+09,9E+09,9E+09]];
    CONST jointtarget jA_v20_t37 := [[89.9999,-49.5,-6,270,8.2,89.9993],[9E+09,9E+09,9E+09,9E+09,9E+09,9E+09]];
    CONST jointtarget jB_v20_t37 := [[44.9994,-58.7,29.3,-90.0002,39.2,-360.001],[9E+09,9E+09,9E+09,9E+09,9E+09,9E+09]];
    CONST jointtarget jBseed_v20_t37 := [[90,-49.5,-6,270,8.2,90],[9E+09,9E+09,9E+09,9E+09,9E+09,9E+09]];
    CONST num seedB_v20_t37 := 30973;

    CONST robtarget rA_v20_t38 := [[1109.24,1191.5,3165.81],[0.640281,-0.168572,0.170881,0.729674],[0,-3,3,0],[9E+09,9E+09,9E+09,9E+09,9E+09,9E+09]];
    CONST robtarget rB_v20_t38 := [[1086.34,1098.89,3130.8],[0.670808,-0.177013,0.11813,0.710442],[0,-3,3,0],[9E+09,9E+09,9E+09,9E+09,9E+09,9E+09]];
    CONST robtarget rB_v20_t38_c7 := [[1086.34,1098.89,3130.8],[0.670808,-0.177013,0.11813,0.710442],[0,-4,4,0],[9E+09,9E+09,9E+09,9E+09,9E+09,9E+09]];
    CONST jointtarget jA_v20_t38 := [[45.0006,20.3,-69.2,-224.999,29.5,270.001],[9E+09,9E+09,9E+09,9E+09,9E+09,9E+09]];
    CONST jointtarget jB_v20_t38 := [[44.9994,-58.7,29.3,-90.0002,39.2,-360.001],[9E+09,9E+09,9E+09,9E+09,9E+09,9E+09]];
    CONST jointtarget jBseed_v20_t38 := [[45,20.3,-69.2,-225,29.5,270],[9E+09,9E+09,9E+09,9E+09,9E+09,9E+09]];
    CONST num seedB_v20_t38 := 29565;

    CONST robtarget rA_v20_t39 := [[1480.92,1480.96,1205.73],[0.225853,-0.371085,0.895843,0.0935498],[0,-1,-1,0],[9E+09,9E+09,9E+09,9E+09,9E+09,9E+09]];
    CONST robtarget rB_v20_t39 := [[1456.28,1484.22,1087.12],[0.226346,-0.426077,0.872501,0.077254],[0,-1,-1,0],[9E+09,9E+09,9E+09,9E+09,9E+09,9E+09]];
    CONST robtarget rB_v20_t39_c5 := [[1456.28,1484.22,1087.12],[0.226346,-0.426077,0.872501,0.077254],[0,0,0,0],[9E+09,9E+09,9E+09,9E+09,9E+09,9E+09]];
    CONST robtarget rB_v20_t39_c8 := [[1456.28,1484.22,1087.12],[0.226346,-0.426077,0.872501,0.077254],[0,0,4,0],[9E+09,9E+09,9E+09,9E+09,9E+09,9E+09]];
    CONST jointtarget jA_v20_t39 := [[45.0008,9.9,13.1,-0.000287096,38.7,-0.000634738],[9E+09,9E+09,9E+09,9E+09,9E+09,9E+09]];
    CONST jointtarget jB_v20_t39 := [[44.9994,-58.7,29.3,-90.0002,39.2,-360.001],[9E+09,9E+09,9E+09,9E+09,9E+09,9E+09]];
    CONST jointtarget jBseed_v20_t39 := [[45,9.9,13.1,0,38.7,0],[9E+09,9E+09,9E+09,9E+09,9E+09,9E+09]];
    CONST num seedB_v20_t39 := 17070;

    CONST robtarget rA_v20_t40 := [[2.59306,1809.58,2287.64],[0.289587,-0.250275,-0.588435,-0.712212],[1,3,2,0],[9E+09,9E+09,9E+09,9E+09,9E+09,9E+09]];
    CONST robtarget rB_v20_t40 := [[58.8918,1754.68,2322.84],[0.27609,-0.33101,-0.530551,-0.729878],[1,3,2,0],[9E+09,9E+09,9E+09,9E+09,9E+09,9E+09]];
    CONST robtarget rB_v20_t40_c9 := [[58.8918,1754.68,2322.84],[0.27609,-0.33101,-0.530551,-0.729878],[0,4,4,0],[9E+09,9E+09,9E+09,9E+09,9E+09,9E+09]];
    CONST jointtarget jA_v20_t40 := [[90.001,-8.2,-2.3,270.001,0.9,225],[9E+09,9E+09,9E+09,9E+09,9E+09,9E+09]];
    CONST jointtarget jB_v20_t40 := [[44.9994,-58.7,29.3,-90.0002,39.2,-360.001],[9E+09,9E+09,9E+09,9E+09,9E+09,9E+09]];
    CONST jointtarget jBseed_v20_t40 := [[90,-8.2,-2.3,270,0.9,225],[9E+09,9E+09,9E+09,9E+09,9E+09,9E+09]];
    CONST num seedB_v20_t40 := 3406;

    CONST robtarget rA_v20_t41 := [[0.0353594,-2007.13,2194.53],[4.37596E-6,-8.3667E-6,0.613596,-0.78962],[-1,-3,1,0],[9E+09,9E+09,9E+09,9E+09,9E+09,9E+09]];
    CONST robtarget rB_v20_t41 := [[22.2989,-2002.94,2292.63],[0.0867015,-0.0345109,-0.548386,0.831003],[-1,-3,1,0],[9E+09,9E+09,9E+09,9E+09,9E+09,9E+09]];
    CONST robtarget rB_v20_t41_c4 := [[22.2989,-2002.94,2292.63],[0.0867015,-0.0345109,-0.548386,0.831003],[0,-4,0,0],[9E+09,9E+09,9E+09,9E+09,9E+09,9E+09]];
    CONST jointtarget jA_v20_t41 := [[-89.999,0.4,-6.5,-180.001,8.2,90.0002],[9E+09,9E+09,9E+09,9E+09,9E+09,9E+09]];
    CONST jointtarget jB_v20_t41 := [[44.9994,-58.7,29.3,-90.0002,39.2,-360.001],[9E+09,9E+09,9E+09,9E+09,9E+09,9E+09]];
    CONST jointtarget jBseed_v20_t41 := [[-90,0.4,-6.5,-180,8.2,90],[9E+09,9E+09,9E+09,9E+09,9E+09,9E+09]];
    CONST num seedB_v20_t41 := 23304;

    CONST robtarget rA_v20_t42 := [[2879.54,-0.0383011,1731.74],[0.683171,0.182419,0.182414,0.683173],[-1,-2,3,0],[9E+09,9E+09,9E+09,9E+09,9E+09,9E+09]];
    CONST robtarget rB_v20_t42 := [[2852.82,-26.2063,1848.27],[0.700158,0.108071,0.180756,0.682222],[-1,-2,3,0],[9E+09,9E+09,9E+09,9E+09,9E+09,9E+09]];
    CONST robtarget rB_v20_t42_c7 := [[2852.82,-26.2063,1848.27],[0.700158,0.108071,0.180756,0.682222],[0,-4,4,0],[9E+09,9E+09,9E+09,9E+09,9E+09,9E+09]];
    CONST jointtarget jA_v20_t42 := [[-0.000761685,58,-62.6,-180,55.5,270.001],[9E+09,9E+09,9E+09,9E+09,9E+09,9E+09]];
    CONST jointtarget jB_v20_t42 := [[44.9994,-58.7,29.3,-90.0002,39.2,-360.001],[9E+09,9E+09,9E+09,9E+09,9E+09,9E+09]];
    CONST jointtarget jBseed_v20_t42 := [[0,58,-62.6,-180,55.5,270],[9E+09,9E+09,9E+09,9E+09,9E+09,9E+09]];
    CONST num seedB_v20_t42 := 25465;

    CONST robtarget rA_v20_t43 := [[-69.7616,-1711.17,1415.04],[0.596096,0.682548,-0.418636,0.0595113],[-1,-1,2,0],[9E+09,9E+09,9E+09,9E+09,9E+09,9E+09]];
    CONST robtarget rB_v20_t43 := [[-71.6267,-1792.33,1516.1],[0.521092,0.733222,-0.430904,0.0719069],[-1,-1,2,0],[9E+09,9E+09,9E+09,9E+09,9E+09,9E+09]];
    CONST robtarget rB_v20_t43_c5 := [[-71.6267,-1792.33,1516.1],[0.521092,0.733222,-0.430904,0.0719069],[0,0,0,0],[9E+09,9E+09,9E+09,9E+09,9E+09,9E+09]];
    CONST jointtarget jA_v20_t43 := [[-89.9993,-14.8,32.9,-89.9994,24.7,225.001],[9E+09,9E+09,9E+09,9E+09,9E+09,9E+09]];
    CONST jointtarget jB_v20_t43 := [[44.9994,-58.7,29.3,-90.0002,39.2,-360.001],[9E+09,9E+09,9E+09,9E+09,9E+09,9E+09]];
    CONST jointtarget jBseed_v20_t43 := [[-90,-14.8,32.9,-90,24.7,225],[9E+09,9E+09,9E+09,9E+09,9E+09,9E+09]];
    CONST num seedB_v20_t43 := 27537;

    CONST robtarget rA_v20_t45 := [[1070.78,38.8497,2959.06],[0.0484453,-0.512485,-0.107518,-0.85056],[0,0,1,0],[9E+09,9E+09,9E+09,9E+09,9E+09,9E+09]];
    CONST robtarget rB_v20_t45 := [[1105.87,-22.8285,3081.32],[0.053535,-0.558759,-0.00749313,-0.827567],[0,0,1,0],[9E+09,9E+09,9E+09,9E+09,9E+09,9E+09]];
    CONST robtarget rB_v20_t45_c5 := [[1105.87,-22.8285,3081.32],[0.053535,-0.558759,-0.00749313,-0.827567],[0,0,0,0],[9E+09,9E+09,9E+09,9E+09,9E+09,9E+09]];
    CONST jointtarget jA_v20_t45 := [[0.000796923,-22,-19.5,45,19.2,135.001],[9E+09,9E+09,9E+09,9E+09,9E+09,9E+09]];
    CONST jointtarget jB_v20_t45 := [[44.9994,-58.7,29.3,-90.0002,39.2,-360.001],[9E+09,9E+09,9E+09,9E+09,9E+09,9E+09]];
    CONST jointtarget jBseed_v20_t45 := [[0,-22,-19.5,45,19.2,135],[9E+09,9E+09,9E+09,9E+09,9E+09,9E+09]];
    CONST num seedB_v20_t45 := 22338;

    CONST robtarget rA_v20_t46 := [[1629.07,91.1358,682.176],[0.234105,-0.835338,-0.469379,-0.164586],[0,0,-4,0],[9E+09,9E+09,9E+09,9E+09,9E+09,9E+09]];
    CONST robtarget rB_v20_t46 := [[1594.18,146.365,730.854],[0.24231,-0.858088,-0.448912,-0.0587325],[0,0,-4,0],[9E+09,9E+09,9E+09,9E+09,9E+09,9E+09]];
    CONST robtarget rB_v20_t46_c2 := [[1594.18,146.365,730.854],[0.24231,-0.858088,-0.448912,-0.0587325],[0,0,-4,0],[9E+09,9E+09,9E+09,9E+09,9E+09,9E+09]];
    CONST jointtarget jA_v20_t46 := [[0.000617197,3.8,41.8,44.9997,50.5,-270.001],[9E+09,9E+09,9E+09,9E+09,9E+09,9E+09]];
    CONST jointtarget jB_v20_t46 := [[44.9994,-58.7,29.3,-90.0002,39.2,-360.001],[9E+09,9E+09,9E+09,9E+09,9E+09,9E+09]];
    CONST jointtarget jBseed_v20_t46 := [[0,3.8,41.8,45,50.5,-270],[9E+09,9E+09,9E+09,9E+09,9E+09,9E+09]];
    CONST num seedB_v20_t46 := 14292;

    CONST robtarget rA_v20_t47 := [[534.731,-663.408,3414.69],[0.89854,0.0107117,-0.314613,0.305826],[-1,2,2,0],[9E+09,9E+09,9E+09,9E+09,9E+09,9E+09]];
    CONST robtarget rB_v20_t47 := [[492.428,-660.667,3367.42],[0.881632,-0.0529796,-0.347455,0.31495],[-1,2,2,0],[9E+09,9E+09,9E+09,9E+09,9E+09,9E+09]];
    CONST robtarget rB_v20_t47_c8 := [[492.428,-660.667,3367.42],[0.881632,-0.0529796,-0.347455,0.31495],[0,0,4,0],[9E+09,9E+09,9E+09,9E+09,9E+09,9E+09]];
    CONST jointtarget jA_v20_t47 := [[-45,6.9,-73.4,225,50.4,225],[9E+09,9E+09,9E+09,9E+09,9E+09,9E+09]];
    CONST jointtarget jB_v20_t47 := [[44.9994,-58.7,29.3,-90.0002,39.2,-360.001],[9E+09,9E+09,9E+09,9E+09,9E+09,9E+09]];
    CONST jointtarget jBseed_v20_t47 := [[-45,6.9,-73.4,225,50.4,225],[9E+09,9E+09,9E+09,9E+09,9E+09,9E+09]];
    CONST num seedB_v20_t47 := 21300;

    CONST robtarget rA_v20_t48 := [[1126.25,-1065.32,3066.07],[0.373313,-0.306767,0.425745,-0.765031],[-1,0,-2,0],[9E+09,9E+09,9E+09,9E+09,9E+09,9E+09]];
    CONST robtarget rB_v20_t48 := [[1150.04,-980.572,3063.64],[0.334908,-0.330321,0.462761,-0.751383],[-1,0,-2,0],[9E+09,9E+09,9E+09,9E+09,9E+09,9E+09]];
    CONST robtarget rB_v20_t48_c5 := [[1150.04,-980.572,3063.64],[0.334908,-0.330321,0.462761,-0.751383],[0,0,0,0],[9E+09,9E+09,9E+09,9E+09,9E+09,9E+09]];
    CONST jointtarget jA_v20_t48 := [[-45,4.9,-48.1,44.9991,21.4,-135],[9E+09,9E+09,9E+09,9E+09,9E+09,9E+09]];
    CONST jointtarget jB_v20_t48 := [[44.9994,-58.7,29.3,-90.0002,39.2,-360.001],[9E+09,9E+09,9E+09,9E+09,9E+09,9E+09]];
    CONST jointtarget jBseed_v20_t48 := [[-45,4.9,-48.1,45,21.4,-135],[9E+09,9E+09,9E+09,9E+09,9E+09,9E+09]];
    CONST num seedB_v20_t48 := 23345;

    CONST robtarget rA_v20_t49 := [[92.6557,2333.67,1846.71],[0.83008,-0.464663,0.205699,-0.229659],[1,2,-4,0],[9E+09,9E+09,9E+09,9E+09,9E+09,9E+09]];
    CONST robtarget rB_v20_t49 := [[170.028,2311.65,1886.9],[0.858303,-0.406772,0.190943,-0.247778],[1,2,-4,0],[9E+09,9E+09,9E+09,9E+09,9E+09,9E+09]];
    CONST robtarget rB_v20_t49_c2 := [[170.028,2311.65,1886.9],[0.858303,-0.406772,0.190943,-0.247778],[0,0,-4,0],[9E+09,9E+09,9E+09,9E+09,9E+09,9E+09]];
    CONST jointtarget jA_v20_t49 := [[90.0004,17.7,-11.4,225.001,51.7,-315.001],[9E+09,9E+09,9E+09,9E+09,9E+09,9E+09]];
    CONST jointtarget jB_v20_t49 := [[44.9994,-58.7,29.3,-90.0002,39.2,-360.001],[9E+09,9E+09,9E+09,9E+09,9E+09,9E+09]];
    CONST jointtarget jBseed_v20_t49 := [[90,17.7,-11.4,225,51.7,-315],[9E+09,9E+09,9E+09,9E+09,9E+09,9E+09]];
    CONST num seedB_v20_t49 := 24043;

    CONST robtarget rA_v20_t50 := [[83.4715,2574.76,2058.06],[0.733111,-0.461026,0.0270302,-0.499272],[1,2,3,0],[9E+09,9E+09,9E+09,9E+09,9E+09,9E+09]];
    CONST robtarget rB_v20_t50 := [[-2.14973,2556.95,1986.66],[0.645181,-0.488867,0.0745097,-0.582408],[1,2,3,0],[9E+09,9E+09,9E+09,9E+09,9E+09,9E+09]];
    CONST robtarget rB_v20_t50_c9 := [[-2.14973,2556.95,1986.66],[0.645181,-0.488867,0.0745097,-0.582408],[0,4,4,0],[9E+09,9E+09,9E+09,9E+09,9E+09,9E+09]];
    CONST jointtarget jA_v20_t50 := [[90.0006,34.2,-40.4,224.999,45,359.999],[9E+09,9E+09,9E+09,9E+09,9E+09,9E+09]];
    CONST jointtarget jB_v20_t50 := [[44.9994,-58.7,29.3,-90.0002,39.2,-360.001],[9E+09,9E+09,9E+09,9E+09,9E+09,9E+09]];
    CONST jointtarget jBseed_v20_t50 := [[90,34.2,-40.4,225,45,360],[9E+09,9E+09,9E+09,9E+09,9E+09,9E+09]];
    CONST num seedB_v20_t50 := 11863;

    CONST robtarget rA_v20_t51 := [[45.3963,-1936.01,1462.72],[0.586538,0.694535,-0.200697,0.365124],[-1,-3,4,0],[9E+09,9E+09,9E+09,9E+09,9E+09,9E+09]];
    CONST robtarget rB_v20_t51 := [[-25.2441,-1889.17,1532.22],[0.650087,0.640966,-0.165024,0.373253],[-1,-3,4,0],[9E+09,9E+09,9E+09,9E+09,9E+09,9E+09]];
    CONST robtarget rB_v20_t51_c7 := [[-25.2441,-1889.17,1532.22],[0.650087,0.640966,-0.165024,0.373253],[0,-4,4,0],[9E+09,9E+09,9E+09,9E+09,9E+09,9E+09]];
    CONST jointtarget jA_v20_t51 := [[-89.9995,-3.7,22.8,-225.001,22.6,360.001],[9E+09,9E+09,9E+09,9E+09,9E+09,9E+09]];
    CONST jointtarget jB_v20_t51 := [[44.9994,-58.7,29.3,-90.0002,39.2,-360.001],[9E+09,9E+09,9E+09,9E+09,9E+09,9E+09]];
    CONST jointtarget jBseed_v20_t51 := [[-90,-3.7,22.8,-225,22.6,360],[9E+09,9E+09,9E+09,9E+09,9E+09,9E+09]];
    CONST num seedB_v20_t51 := 6617;

    CONST robtarget rA_v20_t52 := [[289.849,-416.85,3211.67],[0.84943,0.254078,-0.126982,-0.444734],[-1,2,1,0],[9E+09,9E+09,9E+09,9E+09,9E+09,9E+09]];
    CONST robtarget rB_v20_t52 := [[409.272,-440.589,3202.44],[0.824736,0.247873,-0.0470105,-0.506123],[-1,2,1,0],[9E+09,9E+09,9E+09,9E+09,9E+09,9E+09]];
    CONST robtarget rB_v20_t52_c5 := [[409.272,-440.589,3202.44],[0.824736,0.247873,-0.0470105,-0.506123],[0,0,0,0],[9E+09,9E+09,9E+09,9E+09,9E+09,9E+09]];
    CONST jointtarget jA_v20_t52 := [[-45.0009,-26.4,-29.9,225.001,49.5,134.999],[9E+09,9E+09,9E+09,9E+09,9E+09,9E+09]];
    CONST jointtarget jB_v20_t52 := [[44.9994,-58.7,29.3,-90.0002,39.2,-360.001],[9E+09,9E+09,9E+09,9E+09,9E+09,9E+09]];
    CONST jointtarget jBseed_v20_t52 := [[-45,-26.4,-29.9,225,49.5,135],[9E+09,9E+09,9E+09,9E+09,9E+09,9E+09]];
    CONST num seedB_v20_t52 := 8514;

    CONST robtarget rA_v20_t53 := [[-32.1493,1610.9,3158.36],[0.323958,-0.219353,0.293461,0.872248],[0,0,-1,0],[9E+09,9E+09,9E+09,9E+09,9E+09,9E+09]];
    CONST robtarget rB_v20_t53 := [[-40.0787,1584.03,3146.13],[0.279607,-0.233591,0.265274,0.892684],[0,0,-1,0],[9E+09,9E+09,9E+09,9E+09,9E+09,9E+09]];
    CONST robtarget rB_v20_t53_c5 := [[-40.0787,1584.03,3146.13],[0.279607,-0.233591,0.265274,0.892684],[0,0,0,0],[9E+09,9E+09,9E+09,9E+09,9E+09,9E+09]];
    CONST jointtarget jA_v20_t53 := [[89.9999,15.5,-63.7,89.9997,11.1,-45.0003],[9E+09,9E+09,9E+09,9E+09,9E+09,9E+09]];
    CONST jointtarget jB_v20_t53 := [[44.9994,-58.7,29.3,-90.0002,39.2,-360.001],[9E+09,9E+09,9E+09,9E+09,9E+09,9E+09]];
    CONST jointtarget jBseed_v20_t53 := [[90,15.5,-63.7,90,11.1,-45],[9E+09,9E+09,9E+09,9E+09,9E+09,9E+09]];
    CONST num seedB_v20_t53 := 23755;

    CONST robtarget rA_v20_t54 := [[34.6108,-73.4695,3414.12],[0.670172,0.0922928,0.22554,-0.701059],[0,3,-1,0],[9E+09,9E+09,9E+09,9E+09,9E+09,9E+09]];
    CONST robtarget rB_v20_t54 := [[53.6724,-31.9101,3452.42],[0.612063,0.11164,0.218091,-0.751899],[0,3,-1,0],[9E+09,9E+09,9E+09,9E+09,9E+09,9E+09]];
    CONST robtarget rB_v20_t54_c5 := [[53.6724,-31.9101,3452.42],[0.612063,0.11164,0.218091,-0.751899],[0,0,0,0],[9E+09,9E+09,9E+09,9E+09,9E+09,9E+09]];
    CONST jointtarget jA_v20_t54 := [[0.000642623,-21.8,-57.1,270,26.1,-0.000937495],[9E+09,9E+09,9E+09,9E+09,9E+09,9E+09]];
    CONST jointtarget jB_v20_t54 := [[44.9994,-58.7,29.3,-90.0002,39.2,-360.001],[9E+09,9E+09,9E+09,9E+09,9E+09,9E+09]];
    CONST jointtarget jBseed_v20_t54 := [[0,-21.8,-57.1,270,26.1,0],[9E+09,9E+09,9E+09,9E+09,9E+09,9E+09]];
    CONST num seedB_v20_t54 := 13291;

    CONST robtarget rA_v20_t55 := [[1868.78,42.3039,3020.4],[0.951396,-0.117859,0.279716,0.0520885],[-1,1,-2,0],[9E+09,9E+09,9E+09,9E+09,9E+09,9E+09]];
    CONST robtarget rB_v20_t55 := [[1877.87,19.4159,3039.43],[0.946238,-0.124939,0.295745,0.0394928],[-1,1,-2,0],[9E+09,9E+09,9E+09,9E+09,9E+09,9E+09]];
    CONST robtarget rB_v20_t55_c5 := [[1877.87,19.4159,3039.43],[0.946238,-0.124939,0.295745,0.0394928],[0,0,0,0],[9E+09,9E+09,9E+09,9E+09,9E+09,9E+09]];
    CONST jointtarget jA_v20_t55 := [[-0.000458928,23.8,-66.1,135,21,-135.001],[9E+09,9E+09,9E+09,9E+09,9E+09,9E+09]];
    CONST jointtarget jB_v20_t55 := [[44.9994,-58.7,29.3,-90.0002,39.2,-360.001],[9E+09,9E+09,9E+09,9E+09,9E+09,9E+09]];
    CONST jointtarget jBseed_v20_t55 := [[0,23.8,-66.1,135,21,-135],[9E+09,9E+09,9E+09,9E+09,9E+09,9E+09]];
    CONST num seedB_v20_t55 := 16801;

    CONST robtarget rA_v20_t56 := [[-89.4545,2267.21,473.119],[0.259844,0.101563,-0.894392,-0.349612],[0,-3,-5,0],[9E+09,9E+09,9E+09,9E+09,9E+09,9E+09]];
    CONST robtarget rB_v20_t56 := [[-41.0412,2205.16,446.762],[0.310201,0.0886253,-0.885718,-0.333803],[0,-3,-5,0],[9E+09,9E+09,9E+09,9E+09,9E+09,9E+09]];
    CONST robtarget rB_v20_t56_c1 := [[-41.0412,2205.16,446.762],[0.310201,0.0886253,-0.885718,-0.333803],[0,-4,-4,0],[9E+09,9E+09,9E+09,9E+09,9E+09,9E+09]];
    CONST jointtarget jA_v20_t56 := [[89.9993,35.8,11.5,-269.999,32.4,-360],[9E+09,9E+09,9E+09,9E+09,9E+09,9E+09]];
    CONST jointtarget jB_v20_t56 := [[44.9994,-58.7,29.3,-90.0002,39.2,-360.001],[9E+09,9E+09,9E+09,9E+09,9E+09,9E+09]];
    CONST jointtarget jBseed_v20_t56 := [[90,35.8,11.5,-270,32.4,-360],[9E+09,9E+09,9E+09,9E+09,9E+09,9E+09]];
    CONST num seedB_v20_t56 := 204;

    CONST robtarget rA_v20_t57 := [[977.996,-929.147,3252.22],[0.658607,0.23415,0.098432,0.708323],[-1,1,0,0],[9E+09,9E+09,9E+09,9E+09,9E+09,9E+09]];
    CONST robtarget rB_v20_t57 := [[916.428,-981.258,3190.41],[0.700275,0.226845,0.0641377,0.673826],[-1,1,0,0],[9E+09,9E+09,9E+09,9E+09,9E+09,9E+09]];
    CONST robtarget rB_v20_t57_c5 := [[916.428,-981.258,3190.41],[0.700275,0.226845,0.0641377,0.673826],[0,0,0,0],[9E+09,9E+09,9E+09,9E+09,9E+09,9E+09]];
    CONST jointtarget jA_v20_t57 := [[-44.9993,6.6,-57.3,135,17,0.00078909],[9E+09,9E+09,9E+09,9E+09,9E+09,9E+09]];
    CONST jointtarget jB_v20_t57 := [[44.9994,-58.7,29.3,-90.0002,39.2,-360.001],[9E+09,9E+09,9E+09,9E+09,9E+09,9E+09]];
    CONST jointtarget jBseed_v20_t57 := [[-45,6.6,-57.3,135,17,0],[9E+09,9E+09,9E+09,9E+09,9E+09,9E+09]];
    CONST num seedB_v20_t57 := 28551;

    CONST robtarget rA_v20_t58 := [[-123.329,443.46,2588.5],[0.838458,-0.188136,-0.48,-0.176617],[1,1,1,0],[9E+09,9E+09,9E+09,9E+09,9E+09,9E+09]];
    CONST robtarget rB_v20_t58 := [[-87.1032,422.914,2654.39],[0.886257,-0.173403,-0.413396,-0.116549],[1,1,1,0],[9E+09,9E+09,9E+09,9E+09,9E+09,9E+09]];
    CONST robtarget rB_v20_t58_c4 := [[-87.1032,422.914,2654.39],[0.886257,-0.173403,-0.413396,-0.116549],[0,-4,0,0],[9E+09,9E+09,9E+09,9E+09,9E+09,9E+09]];
    CONST robtarget rB_v20_t58_c5 := [[-87.1032,422.914,2654.39],[0.886257,-0.173403,-0.413396,-0.116549],[0,0,0,0],[9E+09,9E+09,9E+09,9E+09,9E+09,9E+09]];
    CONST jointtarget jA_v20_t58 := [[90.0009,-56.3,12.3,90.0001,47.6,135.001],[9E+09,9E+09,9E+09,9E+09,9E+09,9E+09]];
    CONST jointtarget jB_v20_t58 := [[44.9994,-58.7,29.3,-90.0002,39.2,-360.001],[9E+09,9E+09,9E+09,9E+09,9E+09,9E+09]];
    CONST jointtarget jBseed_v20_t58 := [[90,-56.3,12.3,90,47.6,135],[9E+09,9E+09,9E+09,9E+09,9E+09,9E+09]];
    CONST num seedB_v20_t58 := 14369;

    CONST robtarget rA_v20_t59 := [[-1471.5,-1376.2,2788.02],[0.454771,-0.283495,-0.207828,0.818304],[-2,-2,0,0],[9E+09,9E+09,9E+09,9E+09,9E+09,9E+09]];
    CONST robtarget rB_v20_t59 := [[-1437.55,-1454.8,2817.18],[0.398959,-0.255438,-0.284879,0.833323],[-2,-2,0,0],[9E+09,9E+09,9E+09,9E+09,9E+09,9E+09]];
    CONST robtarget rB_v20_t59_c5 := [[-1437.55,-1454.8,2817.18],[0.398959,-0.255438,-0.284879,0.833323],[0,0,0,0],[9E+09,9E+09,9E+09,9E+09,9E+09,9E+09]];
    CONST jointtarget jA_v20_t59 := [[-135,18.4,-47.6,-135,34.8,44.9997],[9E+09,9E+09,9E+09,9E+09,9E+09,9E+09]];
    CONST jointtarget jB_v20_t59 := [[44.9994,-58.7,29.3,-90.0002,39.2,-360.001],[9E+09,9E+09,9E+09,9E+09,9E+09,9E+09]];
    CONST jointtarget jBseed_v20_t59 := [[-135,18.4,-47.6,-135,34.8,45],[9E+09,9E+09,9E+09,9E+09,9E+09,9E+09]];
    CONST num seedB_v20_t59 := 27176;

    CONST robtarget rA_v20_t60 := [[-887.591,-966.026,3316.83],[0.321453,0.0484874,-0.306999,0.894466],[-2,-3,1,0],[9E+09,9E+09,9E+09,9E+09,9E+09,9E+09]];
    CONST robtarget rB_v20_t60 := [[-866.812,-972.129,3313.35],[0.281221,0.0259898,-0.229979,0.931316],[-2,-3,1,0],[9E+09,9E+09,9E+09,9E+09,9E+09,9E+09]];
    CONST robtarget rB_v20_t60_c4 := [[-866.812,-972.129,3313.35],[0.281221,0.0259898,-0.229979,0.931316],[0,-4,0,0],[9E+09,9E+09,9E+09,9E+09,9E+09,9E+09]];
    CONST jointtarget jA_v20_t60 := [[-135,14.4,-73.2,-269.999,19.4,180],[9E+09,9E+09,9E+09,9E+09,9E+09,9E+09]];
    CONST jointtarget jB_v20_t60 := [[44.9994,-58.7,29.3,-90.0002,39.2,-360.001],[9E+09,9E+09,9E+09,9E+09,9E+09,9E+09]];
    CONST jointtarget jBseed_v20_t60 := [[-135,14.4,-73.2,-270,19.4,180],[9E+09,9E+09,9E+09,9E+09,9E+09,9E+09]];
    CONST num seedB_v20_t60 := 30305;

    CONST robtarget rA_v20_t61 := [[880.753,880.762,2169.96],[0.49504,-0.323117,0.780055,0.205051],[0,0,3,0],[9E+09,9E+09,9E+09,9E+09,9E+09,9E+09]];
    CONST robtarget rB_v20_t61 := [[940.17,957.861,2174.18],[0.502394,-0.290793,0.756195,0.302008],[0,0,3,0],[9E+09,9E+09,9E+09,9E+09,9E+09,9E+09]];
    CONST robtarget rB_v20_t61_c8 := [[940.17,957.861,2174.18],[0.502394,-0.290793,0.756195,0.302008],[0,0,4,0],[9E+09,9E+09,9E+09,9E+09,9E+09,9E+09]];
    CONST jointtarget jA_v20_t61 := [[45.0003,-35,17.6,6.25353E-5,42.6,359.999],[9E+09,9E+09,9E+09,9E+09,9E+09,9E+09]];
    CONST jointtarget jB_v20_t61 := [[44.9994,-58.7,29.3,-90.0002,39.2,-360.001],[9E+09,9E+09,9E+09,9E+09,9E+09,9E+09]];
    CONST jointtarget jBseed_v20_t61 := [[45,-35,17.6,0,42.6,360],[9E+09,9E+09,9E+09,9E+09,9E+09,9E+09]];
    CONST num seedB_v20_t61 := 836;

    CONST robtarget rA_v20_t62 := [[1773.68,-1773.65,1555.59],[9.8816E-7,-0.302747,0.302744,-0.903709],[-1,2,0,0],[9E+09,9E+09,9E+09,9E+09,9E+09,9E+09]];
    CONST robtarget rB_v20_t62 := [[1747.92,-1757.47,1628.22],[0.034584,0.316477,-0.214222,0.923447],[-1,2,0,0],[9E+09,9E+09,9E+09,9E+09,9E+09,9E+09]];
    CONST robtarget rB_v20_t62_c5 := [[1747.92,-1757.47,1628.22],[0.034584,0.316477,-0.214222,0.923447],[0,0,0,0],[9E+09,9E+09,9E+09,9E+09,9E+09,9E+09]];
    CONST jointtarget jA_v20_t62 := [[-44.9995,27.3,-12,180,54.6,44.9996],[9E+09,9E+09,9E+09,9E+09,9E+09,9E+09]];
    CONST jointtarget jB_v20_t62 := [[44.9994,-58.7,29.3,-90.0002,39.2,-360.001],[9E+09,9E+09,9E+09,9E+09,9E+09,9E+09]];
    CONST jointtarget jBseed_v20_t62 := [[-45,27.3,-12,180,54.6,45],[9E+09,9E+09,9E+09,9E+09,9E+09,9E+09]];
    CONST num seedB_v20_t62 := 4477;

    CONST robtarget rA_v20_t63 := [[-138.421,-1830.4,-34.9764],[0.463298,-0.0758695,-0.871343,0.14269],[-1,3,4,0],[9E+09,9E+09,9E+09,9E+09,9E+09,9E+09]];
    CONST robtarget rB_v20_t63 := [[-142.69,-1930.96,-32.5068],[0.542587,-0.00997266,-0.82029,0.180624],[-1,3,4,0],[9E+09,9E+09,9E+09,9E+09,9E+09,9E+09]];
    CONST robtarget rB_v20_t63_c9 := [[-142.69,-1930.96,-32.5068],[0.542587,-0.00997266,-0.82029,0.180624],[0,4,4,0],[9E+09,9E+09,9E+09,9E+09,9E+09,9E+09]];
    CONST jointtarget jA_v20_t63 := [[-89.9991,45.4,26,270.001,56,360],[9E+09,9E+09,9E+09,9E+09,9E+09,9E+09]];
    CONST jointtarget jB_v20_t63 := [[44.9994,-58.7,29.3,-90.0002,39.2,-360.001],[9E+09,9E+09,9E+09,9E+09,9E+09,9E+09]];
    CONST jointtarget jBseed_v20_t63 := [[-90,45.4,26,270,56,360],[9E+09,9E+09,9E+09,9E+09,9E+09,9E+09]];
    CONST num seedB_v20_t63 := 1456;

    CONST robtarget rA_v20_t64 := [[671.82,671.807,-414.537],[0.172244,0.825005,0.341728,-0.415837],[0,-1,1,0],[9E+09,9E+09,9E+09,9E+09,9E+09,9E+09]];
    CONST robtarget rB_v20_t64 := [[578.802,600.885,-396.451],[0.195168,0.788878,0.388868,-0.434009],[0,-1,1,0],[9E+09,9E+09,9E+09,9E+09,9E+09,9E+09]];
    CONST robtarget rB_v20_t64_c5 := [[578.802,600.885,-396.451],[0.195168,0.788878,0.388868,-0.434009],[0,0,0,0],[9E+09,9E+09,9E+09,9E+09,9E+09,9E+09]];
    CONST jointtarget jA_v20_t64 := [[44.9995,59.9,45,-0.000382773,38.6,180],[9E+09,9E+09,9E+09,9E+09,9E+09,9E+09]];
    CONST jointtarget jB_v20_t64 := [[44.9994,-58.7,29.3,-90.0002,39.2,-360.001],[9E+09,9E+09,9E+09,9E+09,9E+09,9E+09]];
    CONST jointtarget jBseed_v20_t64 := [[45,59.9,45,0,38.6,180],[9E+09,9E+09,9E+09,9E+09,9E+09,9E+09]];
    CONST num seedB_v20_t64 := 6934;

    CONST robtarget rA_v20_t66 := [[2428.44,89.7469,626.615],[0.278539,0.22337,0.848882,0.389771],[0,-3,-1,0],[9E+09,9E+09,9E+09,9E+09,9E+09,9E+09]];
    CONST robtarget rB_v20_t66 := [[2345.18,50.7745,609.996],[0.282863,0.236377,0.851732,0.372381],[0,-3,-1,0],[9E+09,9E+09,9E+09,9E+09,9E+09,9E+09]];
    CONST robtarget rB_v20_t66_c4 := [[2345.18,50.7745,609.996],[0.282863,0.236377,0.851732,0.372381],[0,-4,0,0],[9E+09,9E+09,9E+09,9E+09,9E+09,9E+09]];
    CONST jointtarget jA_v20_t66 := [[0.000421927,37.7,2.2,-269.999,32.5,-45.0007],[9E+09,9E+09,9E+09,9E+09,9E+09,9E+09]];
    CONST jointtarget jB_v20_t66 := [[44.9994,-58.7,29.3,-90.0002,39.2,-360.001],[9E+09,9E+09,9E+09,9E+09,9E+09,9E+09]];
    CONST jointtarget jBseed_v20_t66 := [[0,37.7,2.2,-270,32.5,-45],[9E+09,9E+09,9E+09,9E+09,9E+09,9E+09]];
    CONST num seedB_v20_t66 := 23055;

    CONST robtarget rA_v20_t67 := [[-0.0348609,2565.58,2364.53],[0.904846,-0.186559,-0.0772814,-0.374802],[1,-3,-4,0],[9E+09,9E+09,9E+09,9E+09,9E+09,9E+09]];
    CONST robtarget rB_v20_t67 := [[78.4144,2563.56,2337.49],[0.893392,-0.229089,-0.0500607,-0.383228],[1,-3,-4,0],[9E+09,9E+09,9E+09,9E+09,9E+09,9E+09]];
    CONST robtarget rB_v20_t67_c1 := [[78.4144,2563.56,2337.49],[0.893392,-0.229089,-0.0500607,-0.383228],[0,-4,-4,0],[9E+09,9E+09,9E+09,9E+09,9E+09,9E+09]];
    CONST jointtarget jA_v20_t67 := [[90.0008,48.6,-72.1,-180,43.2,-315.001],[9E+09,9E+09,9E+09,9E+09,9E+09,9E+09]];
    CONST jointtarget jB_v20_t67 := [[44.9994,-58.7,29.3,-90.0002,39.2,-360.001],[9E+09,9E+09,9E+09,9E+09,9E+09,9E+09]];
    CONST jointtarget jBseed_v20_t67 := [[90,48.6,-72.1,-180,43.2,-315],[9E+09,9E+09,9E+09,9E+09,9E+09,9E+09]];
    CONST num seedB_v20_t67 := 2893;

    CONST robtarget rA_v20_t68 := [[87.3327,-2777.38,1323.99],[0.422584,0.489571,0.753772,-0.116497],[-2,0,3,0],[9E+09,9E+09,9E+09,9E+09,9E+09,9E+09]];
    CONST robtarget rB_v20_t68 := [[174.87,-2816.94,1334.69],[0.378322,0.495073,0.774495,-0.109236],[-2,0,3,0],[9E+09,9E+09,9E+09,9E+09,9E+09,9E+09]];
    CONST robtarget rB_v20_t68_c8 := [[174.87,-2816.94,1334.69],[0.378322,0.495073,0.774495,-0.109236],[0,0,4,0],[9E+09,9E+09,9E+09,9E+09,9E+09,9E+09]];
    CONST jointtarget jA_v20_t68 := [[-90.0002,45.5,-37.1,45,47.7,315],[9E+09,9E+09,9E+09,9E+09,9E+09,9E+09]];
    CONST jointtarget jB_v20_t68 := [[44.9994,-58.7,29.3,-90.0002,39.2,-360.001],[9E+09,9E+09,9E+09,9E+09,9E+09,9E+09]];
    CONST jointtarget jBseed_v20_t68 := [[-90,45.5,-37.1,45,47.7,315],[9E+09,9E+09,9E+09,9E+09,9E+09,9E+09]];
    CONST num seedB_v20_t68 := 11032;

    CONST robtarget rA_v20_t69 := [[1775.87,1743.47,222.055],[0.353426,-0.33396,0.870444,0.0767409],[0,-1,0,0],[9E+09,9E+09,9E+09,9E+09,9E+09,9E+09]];
    CONST robtarget rB_v20_t69 := [[1726.16,1829.19,316.132],[0.369526,-0.323046,0.868762,0.0659132],[0,-1,0,0],[9E+09,9E+09,9E+09,9E+09,9E+09,9E+09]];
    CONST robtarget rB_v20_t69_c5 := [[1726.16,1829.19,316.132],[0.369526,-0.323046,0.868762,0.0659132],[0,0,0,0],[9E+09,9E+09,9E+09,9E+09,9E+09,9E+09]];
    CONST jointtarget jA_v20_t69 := [[45.0009,51.6,-3.4,-89.9994,7.9,89.9993],[9E+09,9E+09,9E+09,9E+09,9E+09,9E+09]];
    CONST jointtarget jB_v20_t69 := [[44.9994,-58.7,29.3,-90.0002,39.2,-360.001],[9E+09,9E+09,9E+09,9E+09,9E+09,9E+09]];
    CONST jointtarget jBseed_v20_t69 := [[45,51.6,-3.4,-90,7.9,90],[9E+09,9E+09,9E+09,9E+09,9E+09,9E+09]];
    CONST num seedB_v20_t69 := 7220;

    CONST robtarget rA_v20_t71 := [[1804.68,1685.48,2478.72],[0.817526,0.0186524,0.541911,0.194003],[0,-1,-3,0],[9E+09,9E+09,9E+09,9E+09,9E+09,9E+09]];
    CONST robtarget rB_v20_t71 := [[1815.21,1631.88,2450.84],[0.83595,0.000631298,0.460136,0.299102],[0,-1,-3,0],[9E+09,9E+09,9E+09,9E+09,9E+09,9E+09]];
    CONST robtarget rB_v20_t71_c2 := [[1815.21,1631.88,2450.84],[0.83595,0.000631298,0.460136,0.299102],[0,0,-4,0],[9E+09,9E+09,9E+09,9E+09,9E+09,9E+09]];
    CONST jointtarget jA_v20_t71 := [[44.9994,42.5,-71,-89.9991,30.3,-269.999],[9E+09,9E+09,9E+09,9E+09,9E+09,9E+09]];
    CONST jointtarget jB_v20_t71 := [[44.9994,-58.7,29.3,-90.0002,39.2,-360.001],[9E+09,9E+09,9E+09,9E+09,9E+09,9E+09]];
    CONST jointtarget jBseed_v20_t71 := [[45,42.5,-71,-90,30.3,-270],[9E+09,9E+09,9E+09,9E+09,9E+09,9E+09]];
    CONST num seedB_v20_t71 := 14765;

    CONST robtarget rA_v20_t72 := [[305.611,305.605,2786.83],[0.638872,-0.27643,0.66738,0.264636],[0,0,4,0],[9E+09,9E+09,9E+09,9E+09,9E+09,9E+09]];
    CONST robtarget rB_v20_t72 := [[290.018,214.331,2829.22],[0.584476,-0.360377,0.68058,0.255591],[0,0,4,0],[9E+09,9E+09,9E+09,9E+09,9E+09,9E+09]];
    CONST robtarget rB_v20_t72_c8 := [[290.018,214.331,2829.22],[0.584476,-0.360377,0.68058,0.255591],[0,0,4,0],[9E+09,9E+09,9E+09,9E+09,9E+09,9E+09]];
    CONST jointtarget jA_v20_t72 := [[44.9992,-47,-6.3,0.000931642,55.8,360],[9E+09,9E+09,9E+09,9E+09,9E+09,9E+09]];
    CONST jointtarget jB_v20_t72 := [[44.9994,-58.7,29.3,-90.0002,39.2,-360.001],[9E+09,9E+09,9E+09,9E+09,9E+09,9E+09]];
    CONST jointtarget jBseed_v20_t72 := [[45,-47,-6.3,0,55.8,360],[9E+09,9E+09,9E+09,9E+09,9E+09,9E+09]];
    CONST num seedB_v20_t72 := 1011;

    CONST robtarget rA_v20_t73 := [[-631.807,680.494,2445.76],[0.376069,-0.435736,0.276914,0.769431],[1,2,-3,0],[9E+09,9E+09,9E+09,9E+09,9E+09,9E+09]];
    CONST robtarget rB_v20_t73 := [[-614.031,735.051,2376.54],[0.45363,-0.403773,0.227497,0.761204],[1,2,-3,0],[9E+09,9E+09,9E+09,9E+09,9E+09,9E+09]];
    CONST robtarget rB_v20_t73_c2 := [[-614.031,735.051,2376.54],[0.45363,-0.403773,0.227497,0.761204],[0,0,-4,0],[9E+09,9E+09,9E+09,9E+09,9E+09,9E+09]];
    CONST jointtarget jA_v20_t73 := [[135.001,-45.6,17.1,270,11.9,-269.999],[9E+09,9E+09,9E+09,9E+09,9E+09,9E+09]];
    CONST jointtarget jB_v20_t73 := [[44.9994,-58.7,29.3,-90.0002,39.2,-360.001],[9E+09,9E+09,9E+09,9E+09,9E+09,9E+09]];
    CONST jointtarget jBseed_v20_t73 := [[135,-45.6,17.1,270,11.9,-270],[9E+09,9E+09,9E+09,9E+09,9E+09,9E+09]];
    CONST num seedB_v20_t73 := 27326;

    CONST robtarget rA_v20_t74 := [[-0.0164144,2575.33,263.536],[0.553392,-0.832921,-5.89033E-6,2.82977E-6],[1,1,1,0],[9E+09,9E+09,9E+09,9E+09,9E+09,9E+09]];
    CONST robtarget rB_v20_t74 := [[20.299,2604.83,326.135],[0.508698,-0.859512,-0.033008,0.0370937],[1,1,1,0],[9E+09,9E+09,9E+09,9E+09,9E+09,9E+09]];
    CONST robtarget rB_v20_t74_c5 := [[20.299,2604.83,326.135],[0.508698,-0.859512,-0.033008,0.0370937],[0,0,0,0],[9E+09,9E+09,9E+09,9E+09,9E+09,9E+09]];
    CONST jointtarget jA_v20_t74 := [[90.0003,53.9,-6.6,179.999,24.5,90.0005],[9E+09,9E+09,9E+09,9E+09,9E+09,9E+09]];
    CONST jointtarget jB_v20_t74 := [[44.9994,-58.7,29.3,-90.0002,39.2,-360.001],[9E+09,9E+09,9E+09,9E+09,9E+09,9E+09]];
    CONST jointtarget jBseed_v20_t74 := [[90,53.9,-6.6,180,24.5,90],[9E+09,9E+09,9E+09,9E+09,9E+09,9E+09]];
    CONST num seedB_v20_t74 := 10703;

    CONST robtarget rA_v20_t75 := [[496.518,489.512,2649.89],[0.629064,-0.443783,0.013369,-0.638088],[0,-1,-2,0],[9E+09,9E+09,9E+09,9E+09,9E+09,9E+09]];
    CONST robtarget rB_v20_t75 := [[470.913,451.976,2676.81],[0.659942,-0.362913,-0.0117362,-0.657748],[0,-1,-2,0],[9E+09,9E+09,9E+09,9E+09,9E+09,9E+09]];
    CONST robtarget rB_v20_t75_c4 := [[470.913,451.976,2676.81],[0.659942,-0.362913,-0.0117362,-0.657748],[0,-4,0,0],[9E+09,9E+09,9E+09,9E+09,9E+09,9E+09]];
    CONST jointtarget jA_v20_t75 := [[44.9992,-48,9,-44.9999,2.4,-90],[9E+09,9E+09,9E+09,9E+09,9E+09,9E+09]];
    CONST jointtarget jB_v20_t75 := [[44.9994,-58.7,29.3,-90.0002,39.2,-360.001],[9E+09,9E+09,9E+09,9E+09,9E+09,9E+09]];
    CONST jointtarget jBseed_v20_t75 := [[45,-48,9,-45,2.4,-90],[9E+09,9E+09,9E+09,9E+09,9E+09,9E+09]];
    CONST num seedB_v20_t75 := 9575;

    CONST robtarget rA_v20_t76 := [[1203.31,1203.31,207.41],[0.0929016,-0.371242,-0.896238,0.22429],[0,-1,1,0],[9E+09,9E+09,9E+09,9E+09,9E+09,9E+09]];
    CONST robtarget rB_v20_t76 := [[1264.16,1156.3,233.184],[0.0906918,-0.385927,-0.886587,0.238325],[0,-1,1,0],[9E+09,9E+09,9E+09,9E+09,9E+09,9E+09]];
    CONST robtarget rB_v20_t76_c2 := [[1264.16,1156.3,233.184],[0.0906918,-0.385927,-0.886587,0.238325],[0,0,-4,0],[9E+09,9E+09,9E+09,9E+09,9E+09,9E+09]];
    CONST robtarget rB_v20_t76_c5 := [[1264.16,1156.3,233.184],[0.0906918,-0.385927,-0.886587,0.238325],[0,0,0,0],[9E+09,9E+09,9E+09,9E+09,9E+09,9E+09]];
    CONST jointtarget jA_v20_t76 := [[44.9999,30.5,32,-5.51481E-5,55.6,90.0009],[9E+09,9E+09,9E+09,9E+09,9E+09,9E+09]];
    CONST jointtarget jB_v20_t76 := [[44.9994,-58.7,29.3,-90.0002,39.2,-360.001],[9E+09,9E+09,9E+09,9E+09,9E+09,9E+09]];
    CONST jointtarget jBseed_v20_t76 := [[45,30.5,32,0,55.6,90],[9E+09,9E+09,9E+09,9E+09,9E+09,9E+09]];
    CONST num seedB_v20_t76 := 4366;

    CONST robtarget rA_v20_t77 := [[-66.1683,-2707.56,628.87],[0.0680975,0.376565,0.660656,-0.64583],[-1,2,-4,0],[9E+09,9E+09,9E+09,9E+09,9E+09,9E+09]];
    CONST robtarget rB_v20_t77 := [[-157.214,-2767.49,634.27],[0.121004,0.430473,0.656039,-0.608],[-1,2,-4,0],[9E+09,9E+09,9E+09,9E+09,9E+09,9E+09]];
    CONST robtarget rB_v20_t77_c3 := [[-157.214,-2767.49,634.27],[0.121004,0.430473,0.656039,-0.608],[0,4,-4,0],[9E+09,9E+09,9E+09,9E+09,9E+09,9E+09]];
    CONST jointtarget jA_v20_t77 := [[-89.9993,50.1,-14.7,224.999,34.1,-270],[9E+09,9E+09,9E+09,9E+09,9E+09,9E+09]];
    CONST jointtarget jB_v20_t77 := [[44.9994,-58.7,29.3,-90.0002,39.2,-360.001],[9E+09,9E+09,9E+09,9E+09,9E+09,9E+09]];
    CONST jointtarget jBseed_v20_t77 := [[-90,50.1,-14.7,225,34.1,-270],[9E+09,9E+09,9E+09,9E+09,9E+09,9E+09]];
    CONST num seedB_v20_t77 := 7695;

    CONST robtarget rA_v20_t78 := [[-63.8266,-1939.01,476.689],[0.189737,-0.060195,-0.854454,0.479879],[-2,2,0,0],[9E+09,9E+09,9E+09,9E+09,9E+09,9E+09]];
    CONST robtarget rB_v20_t78 := [[-21.8438,-1910,499.858],[0.104117,-0.113076,-0.888092,0.433204],[-2,2,0,0],[9E+09,9E+09,9E+09,9E+09,9E+09,9E+09]];
    CONST robtarget rB_v20_t78_c6 := [[-21.8438,-1910,499.858],[0.104117,-0.113076,-0.888092,0.433204],[0,4,0,0],[9E+09,9E+09,9E+09,9E+09,9E+09,9E+09]];
    CONST jointtarget jA_v20_t78 := [[-90.001,22.6,32.2,224.999,32.7,45.0009],[9E+09,9E+09,9E+09,9E+09,9E+09,9E+09]];
    CONST jointtarget jB_v20_t78 := [[44.9994,-58.7,29.3,-90.0002,39.2,-360.001],[9E+09,9E+09,9E+09,9E+09,9E+09,9E+09]];
    CONST jointtarget jBseed_v20_t78 := [[-90,22.6,32.2,225,32.7,45],[9E+09,9E+09,9E+09,9E+09,9E+09,9E+09]];
    CONST num seedB_v20_t78 := 14839;

    CONST robtarget rA_v20_t79 := [[9.65256,-1927.59,545.781],[0.16516,0.346925,0.863214,-0.327455],[-2,1,-3,0],[9E+09,9E+09,9E+09,9E+09,9E+09,9E+09]];
    CONST robtarget rB_v20_t79 := [[1.20748,-1870.25,555.902],[0.237592,0.299512,0.882323,-0.274498],[-2,1,-3,0],[9E+09,9E+09,9E+09,9E+09,9E+09,9E+09]];
    CONST robtarget rB_v20_t79_c2 := [[1.20748,-1870.25,555.902],[0.237592,0.299512,0.882323,-0.274498],[0,0,-4,0],[9E+09,9E+09,9E+09,9E+09,9E+09,9E+09]];
    CONST jointtarget jA_v20_t79 := [[-90.0007,18.4,32,135,4.7,-180.001],[9E+09,9E+09,9E+09,9E+09,9E+09,9E+09]];
    CONST jointtarget jB_v20_t79 := [[44.9994,-58.7,29.3,-90.0002,39.2,-360.001],[9E+09,9E+09,9E+09,9E+09,9E+09,9E+09]];
    CONST jointtarget jBseed_v20_t79 := [[-90,18.4,32,135,4.7,-180],[9E+09,9E+09,9E+09,9E+09,9E+09,9E+09]];
    CONST num seedB_v20_t79 := 23834;

    CONST robtarget rA_v20_t80 := [[-0.0237289,1591.05,2525.55],[0.414625,-0.572794,0.572778,0.414631],[1,0,3,0],[9E+09,9E+09,9E+09,9E+09,9E+09,9E+09]];
    CONST robtarget rB_v20_t80 := [[-21.3162,1598.81,2592.28],[0.420794,-0.6212,0.550366,0.366251],[1,0,3,0],[9E+09,9E+09,9E+09,9E+09,9E+09,9E+09]];
    CONST robtarget rB_v20_t80_c8 := [[-21.3162,1598.81,2592.28],[0.420794,-0.6212,0.550366,0.366251],[0,0,4,0],[9E+09,9E+09,9E+09,9E+09,9E+09,9E+09]];
    CONST jointtarget jA_v20_t80 := [[90.0008,-11.4,-12.5,0.000654311,42.1,359.999],[9E+09,9E+09,9E+09,9E+09,9E+09,9E+09]];
    CONST jointtarget jB_v20_t80 := [[44.9994,-58.7,29.3,-90.0002,39.2,-360.001],[9E+09,9E+09,9E+09,9E+09,9E+09,9E+09]];
    CONST jointtarget jBseed_v20_t80 := [[90,-11.4,-12.5,0,42.1,360],[9E+09,9E+09,9E+09,9E+09,9E+09,9E+09]];
    CONST num seedB_v20_t80 := 26894;

    CONST robtarget rA_v20_t81 := [[-0.00116063,-1034.26,1675.62],[0.34833,0.855698,0.35444,-0.14429],[-1,-1,-4,0],[9E+09,9E+09,9E+09,9E+09,9E+09,9E+09]];
    CONST robtarget rB_v20_t81 := [[-87.0059,-1004.99,1675.16],[0.313491,0.889431,0.321203,-0.0863956],[-1,-1,-4,0],[9E+09,9E+09,9E+09,9E+09,9E+09,9E+09]];
    CONST robtarget rB_v20_t81_c2 := [[-87.0059,-1004.99,1675.16],[0.313491,0.889431,0.321203,-0.0863956],[0,0,-4,0],[9E+09,9E+09,9E+09,9E+09,9E+09,9E+09]];
    CONST jointtarget jA_v20_t81 := [[-89.9999,-53.1,43.6,-0.000929662,55.2,-315],[9E+09,9E+09,9E+09,9E+09,9E+09,9E+09]];
    CONST jointtarget jB_v20_t81 := [[44.9994,-58.7,29.3,-90.0002,39.2,-360.001],[9E+09,9E+09,9E+09,9E+09,9E+09,9E+09]];
    CONST jointtarget jBseed_v20_t81 := [[-90,-53.1,43.6,0,55.2,-315],[9E+09,9E+09,9E+09,9E+09,9E+09,9E+09]];
    CONST num seedB_v20_t81 := 21865;

    CONST robtarget rA_v20_t82 := [[100.817,1972.33,152.215],[0.338673,0.0710621,0.782423,0.51775],[0,-2,2,0],[9E+09,9E+09,9E+09,9E+09,9E+09,9E+09]];
    CONST robtarget rB_v20_t82 := [[140.198,1995.52,258.125],[0.329362,0.133597,0.71853,0.59782],[0,-2,2,0],[9E+09,9E+09,9E+09,9E+09,9E+09,9E+09]];
    CONST robtarget rB_v20_t82_c4 := [[140.198,1995.52,258.125],[0.329362,0.133597,0.71853,0.59782],[0,-4,0,0],[9E+09,9E+09,9E+09,9E+09,9E+09,9E+09]];
    CONST robtarget rB_v20_t82_c7 := [[140.198,1995.52,258.125],[0.329362,0.133597,0.71853,0.59782],[0,-4,4,0],[9E+09,9E+09,9E+09,9E+09,9E+09,9E+09]];
    CONST jointtarget jA_v20_t82 := [[89.9993,40,26.3,-135,58.6,225],[9E+09,9E+09,9E+09,9E+09,9E+09,9E+09]];
    CONST jointtarget jB_v20_t82 := [[44.9994,-58.7,29.3,-90.0002,39.2,-360.001],[9E+09,9E+09,9E+09,9E+09,9E+09,9E+09]];
    CONST jointtarget jBseed_v20_t82 := [[90,40,26.3,-135,58.6,225],[9E+09,9E+09,9E+09,9E+09,9E+09,9E+09]];
    CONST num seedB_v20_t82 := 27031;

    CONST robtarget rA_v20_t83 := [[1177.44,-1198.06,-9.02825],[0.187405,0.698353,0.689424,-0.0433242],[-1,-2,-2,0],[9E+09,9E+09,9E+09,9E+09,9E+09,9E+09]];
    CONST robtarget rB_v20_t83 := [[1075.19,-1082.99,36.7358],[0.116342,0.703991,0.7006,0.00454125],[-1,-2,-2,0],[9E+09,9E+09,9E+09,9E+09,9E+09,9E+09]];
    CONST robtarget rB_v20_t83_c2 := [[1075.19,-1082.99,36.7358],[0.116342,0.703991,0.7006,0.00454125],[0,0,-4,0],[9E+09,9E+09,9E+09,9E+09,9E+09,9E+09]];
    CONST jointtarget jA_v20_t83 := [[-44.9995,36.4,37,-135.001,7.1,-180],[9E+09,9E+09,9E+09,9E+09,9E+09,9E+09]];
    CONST jointtarget jB_v20_t83 := [[44.9994,-58.7,29.3,-90.0002,39.2,-360.001],[9E+09,9E+09,9E+09,9E+09,9E+09,9E+09]];
    CONST jointtarget jBseed_v20_t83 := [[-45,36.4,37,-135,7.1,-180],[9E+09,9E+09,9E+09,9E+09,9E+09,9E+09]];
    CONST num seedB_v20_t83 := 32003;

    CONST robtarget rA_v20_t85 := [[-671.821,-581.825,2747.93],[0.905972,-0.0596286,-0.31564,0.275737],[-2,-2,3,0],[9E+09,9E+09,9E+09,9E+09,9E+09,9E+09]];
    CONST robtarget rB_v20_t85 := [[-582.893,-632.21,2702.74],[0.94771,-0.0482958,-0.235591,0.209784],[-2,-2,3,0],[9E+09,9E+09,9E+09,9E+09,9E+09,9E+09]];
    CONST robtarget rB_v20_t85_c7 := [[-582.893,-632.21,2702.74],[0.94771,-0.0482958,-0.235591,0.209784],[0,-4,4,0],[9E+09,9E+09,9E+09,9E+09,9E+09,9E+09]];
    CONST robtarget rB_v20_t85_c8 := [[-582.893,-632.21,2702.74],[0.94771,-0.0482958,-0.235591,0.209784],[0,0,4,0],[9E+09,9E+09,9E+09,9E+09,9E+09,9E+09]];
    CONST jointtarget jA_v20_t85 := [[-135.001,-36.7,1.9,-135,32.6,315],[9E+09,9E+09,9E+09,9E+09,9E+09,9E+09]];
    CONST jointtarget jB_v20_t85 := [[44.9994,-58.7,29.3,-90.0002,39.2,-360.001],[9E+09,9E+09,9E+09,9E+09,9E+09,9E+09]];
    CONST jointtarget jBseed_v20_t85 := [[-135,-36.7,1.9,-135,32.6,315],[9E+09,9E+09,9E+09,9E+09,9E+09,9E+09]];
    CONST num seedB_v20_t85 := 22618;

    CONST robtarget rA_v20_t86 := [[-1481.83,1339.66,1674.36],[0.60512,-0.373131,-0.659479,0.244314],[1,-4,1,0],[9E+09,9E+09,9E+09,9E+09,9E+09,9E+09]];
    CONST robtarget rB_v20_t86 := [[-1467.83,1269.76,1699.93],[0.629056,-0.356699,-0.629971,0.28318],[1,-4,1,0],[9E+09,9E+09,9E+09,9E+09,9E+09,9E+09]];
    CONST robtarget rB_v20_t86_c4 := [[-1467.83,1269.76,1699.93],[0.629056,-0.356699,-0.629971,0.28318],[0,-4,0,0],[9E+09,9E+09,9E+09,9E+09,9E+09,9E+09]];
    CONST jointtarget jA_v20_t86 := [[135.001,-0.7,11.4,-270,37,135],[9E+09,9E+09,9E+09,9E+09,9E+09,9E+09]];
    CONST jointtarget jB_v20_t86 := [[44.9994,-58.7,29.3,-90.0002,39.2,-360.001],[9E+09,9E+09,9E+09,9E+09,9E+09,9E+09]];
    CONST jointtarget jBseed_v20_t86 := [[135,-0.7,11.4,-270,37,135],[9E+09,9E+09,9E+09,9E+09,9E+09,9E+09]];
    CONST num seedB_v20_t86 := 24016;

    CONST robtarget rA_v20_t88 := [[2723.72,0.0140555,1763.06],[0.242419,0.664255,0.664249,0.24243],[0,0,1,0],[9E+09,9E+09,9E+09,9E+09,9E+09,9E+09]];
    CONST robtarget rB_v20_t88 := [[2731.33,83.6101,1787.08],[0.232632,0.612533,0.713412,0.248451],[0,0,1,0],[9E+09,9E+09,9E+09,9E+09,9E+09,9E+09]];
    CONST robtarget rB_v20_t88_c5 := [[2731.33,83.6101,1787.08],[0.232632,0.612533,0.713412,0.248451],[0,0,0,0],[9E+09,9E+09,9E+09,9E+09,9E+09,9E+09]];
    CONST jointtarget jA_v20_t88 := [[0.000261722,45.4,-54.2,0.00064797,58.7,90.0006],[9E+09,9E+09,9E+09,9E+09,9E+09,9E+09]];
    CONST jointtarget jB_v20_t88 := [[44.9994,-58.7,29.3,-90.0002,39.2,-360.001],[9E+09,9E+09,9E+09,9E+09,9E+09,9E+09]];
    CONST jointtarget jBseed_v20_t88 := [[0,45.4,-54.2,0,58.7,90],[9E+09,9E+09,9E+09,9E+09,9E+09,9E+09]];
    CONST num seedB_v20_t88 := 30584;

    CONST robtarget rA_v20_t89 := [[851.471,708.931,2946.49],[0.56741,0.318418,0.659866,0.375809],[0,-1,0,0],[9E+09,9E+09,9E+09,9E+09,9E+09,9E+09]];
    CONST robtarget rB_v20_t89 := [[831.444,740.959,3036.01],[0.563014,0.190328,0.693343,0.407511],[0,-1,0,0],[9E+09,9E+09,9E+09,9E+09,9E+09,9E+09]];
    CONST robtarget rB_v20_t89_c5 := [[831.444,740.959,3036.01],[0.563014,0.190328,0.693343,0.407511],[0,0,0,0],[9E+09,9E+09,9E+09,9E+09,9E+09,9E+09]];
    CONST jointtarget jA_v20_t89 := [[45,-16.9,-27,-44.9992,58.6,90],[9E+09,9E+09,9E+09,9E+09,9E+09,9E+09]];
    CONST jointtarget jB_v20_t89 := [[44.9994,-58.7,29.3,-90.0002,39.2,-360.001],[9E+09,9E+09,9E+09,9E+09,9E+09,9E+09]];
    CONST jointtarget jBseed_v20_t89 := [[45,-16.9,-27,-45,58.6,90],[9E+09,9E+09,9E+09,9E+09,9E+09,9E+09]];
    CONST num seedB_v20_t89 := 6372;

    CONST robtarget rA_v20_t90 := [[194.441,0.00189609,3359.76],[0.673444,0.215567,-0.215576,-0.673447],[-1,-3,-3,0],[9E+09,9E+09,9E+09,9E+09,9E+09,9E+09]];
    CONST robtarget rB_v20_t90 := [[155.596,-64.4535,3294.16],[0.606121,0.228098,-0.220384,-0.729397],[-1,-3,-3,0],[9E+09,9E+09,9E+09,9E+09,9E+09,9E+09]];
    CONST robtarget rB_v20_t90_c1 := [[155.596,-64.4535,3294.16],[0.606121,0.228098,-0.220384,-0.729397],[0,-4,-4,0],[9E+09,9E+09,9E+09,9E+09,9E+09,9E+09]];
    CONST robtarget rB_v20_t90_c4 := [[155.596,-64.4535,3294.16],[0.606121,0.228098,-0.220384,-0.729397],[0,-4,0,0],[9E+09,9E+09,9E+09,9E+09,9E+09,9E+09]];
    CONST jointtarget jA_v20_t90 := [[-5.56453E-5,-21.6,-46.8,-180.001,57.1,-270],[9E+09,9E+09,9E+09,9E+09,9E+09,9E+09]];
    CONST jointtarget jB_v20_t90 := [[44.9994,-58.7,29.3,-90.0002,39.2,-360.001],[9E+09,9E+09,9E+09,9E+09,9E+09,9E+09]];
    CONST jointtarget jBseed_v20_t90 := [[0,-21.6,-46.8,-180,57.1,-270],[9E+09,9E+09,9E+09,9E+09,9E+09,9E+09]];
    CONST num seedB_v20_t90 := 6946;

    CONST robtarget rA_v20_t91 := [[1724.99,-47.6347,942.405],[0.336039,0.776712,0.252175,0.469259],[0,2,2,0],[9E+09,9E+09,9E+09,9E+09,9E+09,9E+09]];
    CONST robtarget rB_v20_t91 := [[1776.14,-87.7896,923.615],[0.316804,0.807187,0.318099,0.383273],[0,2,2,0],[9E+09,9E+09,9E+09,9E+09,9E+09,9E+09]];
    CONST robtarget rB_v20_t91_c9 := [[1776.14,-87.7896,923.615],[0.316804,0.807187,0.318099,0.383273],[0,4,4,0],[9E+09,9E+09,9E+09,9E+09,9E+09,9E+09]];
    CONST jointtarget jA_v20_t91 := [[0.000621113,-4.7,42.4,225,23.8,270],[9E+09,9E+09,9E+09,9E+09,9E+09,9E+09]];
    CONST jointtarget jB_v20_t91 := [[44.9994,-58.7,29.3,-90.0002,39.2,-360.001],[9E+09,9E+09,9E+09,9E+09,9E+09,9E+09]];
    CONST jointtarget jBseed_v20_t91 := [[0,-4.7,42.4,225,23.8,270],[9E+09,9E+09,9E+09,9E+09,9E+09,9E+09]];
    CONST num seedB_v20_t91 := 23033;

    CONST robtarget rA_v20_t92 := [[-34.1148,-2190.55,2380.74],[0.220537,0.336001,0.595903,-0.695245],[-1,-1,-5,0],[9E+09,9E+09,9E+09,9E+09,9E+09,9E+09]];
    CONST robtarget rB_v20_t92 := [[0.606609,-2100.58,2475.48],[0.147437,0.392201,0.567615,-0.708699],[-1,-1,-5,0],[9E+09,9E+09,9E+09,9E+09,9E+09,9E+09]];
    CONST robtarget rB_v20_t92_c2 := [[0.606609,-2100.58,2475.48],[0.147437,0.392201,0.567615,-0.708699],[0,0,-4,0],[9E+09,9E+09,9E+09,9E+09,9E+09,9E+09]];
    CONST jointtarget jA_v20_t92 := [[-89.9996,14.1,-29.9,-45.0001,16.8,-360],[9E+09,9E+09,9E+09,9E+09,9E+09,9E+09]];
    CONST jointtarget jB_v20_t92 := [[44.9994,-58.7,29.3,-90.0002,39.2,-360.001],[9E+09,9E+09,9E+09,9E+09,9E+09,9E+09]];
    CONST jointtarget jBseed_v20_t92 := [[-90,14.1,-29.9,-45,16.8,-360],[9E+09,9E+09,9E+09,9E+09,9E+09,9E+09]];
    CONST num seedB_v20_t92 := 5875;

    CONST robtarget rA_v20_t93 := [[-1072.72,1072.74,2779.33],[0.780924,-0.493677,-0.204488,0.323458],[1,-1,-2,0],[9E+09,9E+09,9E+09,9E+09,9E+09,9E+09]];
    CONST robtarget rB_v20_t93 := [[-962.821,1044.05,2810.85],[0.817171,-0.405499,-0.26636,0.311215],[1,-1,-2,0],[9E+09,9E+09,9E+09,9E+09,9E+09,9E+09]];
    CONST robtarget rB_v20_t93_c2 := [[-962.821,1044.05,2810.85],[0.817171,-0.405499,-0.26636,0.311215],[0,0,-4,0],[9E+09,9E+09,9E+09,9E+09,9E+09,9E+09]];
    CONST robtarget rB_v20_t93_c5 := [[-962.821,1044.05,2810.85],[0.817171,-0.405499,-0.26636,0.311215],[0,0,0,0],[9E+09,9E+09,9E+09,9E+09,9E+09,9E+09]];
    CONST jointtarget jA_v20_t93 := [[134.999,-10.4,-19.1,-0.000457001,4.1,-90.0003],[9E+09,9E+09,9E+09,9E+09,9E+09,9E+09]];
    CONST jointtarget jB_v20_t93 := [[44.9994,-58.7,29.3,-90.0002,39.2,-360.001],[9E+09,9E+09,9E+09,9E+09,9E+09,9E+09]];
    CONST jointtarget jBseed_v20_t93 := [[135,-10.4,-19.1,0,4.1,-90],[9E+09,9E+09,9E+09,9E+09,9E+09,9E+09]];
    CONST num seedB_v20_t93 := 19718;

    CONST robtarget rA_v20_t94 := [[1261.8,1288.91,2909.94],[0.605786,-0.0509351,0.464842,0.6437],[0,-3,3,0],[9E+09,9E+09,9E+09,9E+09,9E+09,9E+09]];
    CONST robtarget rB_v20_t94 := [[1284.69,1248.02,2925.87],[0.602081,-0.130204,0.500402,0.608394],[0,-3,3,0],[9E+09,9E+09,9E+09,9E+09,9E+09,9E+09]];
    CONST robtarget rB_v20_t94_c7 := [[1284.69,1248.02,2925.87],[0.602081,-0.130204,0.500402,0.608394],[0,-4,4,0],[9E+09,9E+09,9E+09,9E+09,9E+09,9E+09]];
    CONST jointtarget jA_v20_t94 := [[44.9994,9.5,-44,-269.999,6.6,315],[9E+09,9E+09,9E+09,9E+09,9E+09,9E+09]];
    CONST jointtarget jB_v20_t94 := [[44.9994,-58.7,29.3,-90.0002,39.2,-360.001],[9E+09,9E+09,9E+09,9E+09,9E+09,9E+09]];
    CONST jointtarget jBseed_v20_t94 := [[45,9.5,-44,-270,6.6,315],[9E+09,9E+09,9E+09,9E+09,9E+09,9E+09]];
    CONST num seedB_v20_t94 := 30560;

    CONST robtarget rA_v20_t95 := [[-961.313,1074.32,3209.46],[0.617087,-0.240586,-0.0856945,-0.744297],[1,2,2,0],[9E+09,9E+09,9E+09,9E+09,9E+09,9E+09]];
    CONST robtarget rB_v20_t95 := [[-965.959,1093.4,3199.69],[0.673111,-0.172048,-0.107609,-0.711155],[1,2,2,0],[9E+09,9E+09,9E+09,9E+09,9E+09,9E+09]];
    CONST robtarget rB_v20_t95_c8 := [[-965.959,1093.4,3199.69],[0.673111,-0.172048,-0.107609,-0.711155],[0,0,4,0],[9E+09,9E+09,9E+09,9E+09,9E+09,9E+09]];
    CONST jointtarget jA_v20_t95 := [[135.001,12.1,-61.1,224.999,42.6,270],[9E+09,9E+09,9E+09,9E+09,9E+09,9E+09]];
    CONST jointtarget jB_v20_t95 := [[44.9994,-58.7,29.3,-90.0002,39.2,-360.001],[9E+09,9E+09,9E+09,9E+09,9E+09,9E+09]];
    CONST jointtarget jBseed_v20_t95 := [[135,12.1,-61.1,225,42.6,270],[9E+09,9E+09,9E+09,9E+09,9E+09,9E+09]];
    CONST num seedB_v20_t95 := 8333;

    CONST robtarget rA_v20_t96 := [[-320.998,254.398,3485.08],[0.713719,0.142629,0.00806667,-0.685709],[1,1,4,0],[9E+09,9E+09,9E+09,9E+09,9E+09,9E+09]];
    CONST robtarget rB_v20_t96 := [[-343.396,267.266,3451.91],[0.656227,0.112196,-0.0646713,-0.743368],[1,1,4,0],[9E+09,9E+09,9E+09,9E+09,9E+09,9E+09]];
    CONST robtarget rB_v20_t96_c8 := [[-343.396,267.266,3451.91],[0.656227,0.112196,-0.0646713,-0.743368],[0,0,4,0],[9E+09,9E+09,9E+09,9E+09,9E+09,9E+09]];
    CONST jointtarget jA_v20_t96 := [[135.001,-7.1,-67.1,135,23.5,360],[9E+09,9E+09,9E+09,9E+09,9E+09,9E+09]];
    CONST jointtarget jB_v20_t96 := [[44.9994,-58.7,29.3,-90.0002,39.2,-360.001],[9E+09,9E+09,9E+09,9E+09,9E+09,9E+09]];
    CONST jointtarget jBseed_v20_t96 := [[135,-7.1,-67.1,135,23.5,360],[9E+09,9E+09,9E+09,9E+09,9E+09,9E+09]];
    CONST num seedB_v20_t96 := 28270;

    CONST robtarget rA_v20_t97 := [[40.3755,-194.07,3407.12],[0.876125,0.23443,-0.275773,0.318428],[-1,2,1,0],[9E+09,9E+09,9E+09,9E+09,9E+09,9E+09]];
    CONST robtarget rB_v20_t97 := [[24.2871,-147.924,3461.13],[0.914722,0.234561,-0.195349,0.264771],[-1,2,1,0],[9E+09,9E+09,9E+09,9E+09,9E+09,9E+09]];
    CONST robtarget rB_v20_t97_c6 := [[24.2871,-147.924,3461.13],[0.914722,0.234561,-0.195349,0.264771],[0,4,0,0],[9E+09,9E+09,9E+09,9E+09,9E+09,9E+09]];
    CONST jointtarget jA_v20_t97 := [[-44.9998,-18.4,-58,269.999,40.6,179.999],[9E+09,9E+09,9E+09,9E+09,9E+09,9E+09]];
    CONST jointtarget jB_v20_t97 := [[44.9994,-58.7,29.3,-90.0002,39.2,-360.001],[9E+09,9E+09,9E+09,9E+09,9E+09,9E+09]];
    CONST jointtarget jBseed_v20_t97 := [[-45,-18.4,-58,270,40.6,180],[9E+09,9E+09,9E+09,9E+09,9E+09,9E+09]];
    CONST num seedB_v20_t97 := 1725;

    CONST robtarget rA_v20_t98 := [[-1185.61,1125.65,2560.61],[0.379423,0.313029,-0.480689,-0.72594],[1,0,-5,0],[9E+09,9E+09,9E+09,9E+09,9E+09,9E+09]];
    CONST robtarget rB_v20_t98 := [[-1181.81,1033.32,2627.22],[0.332817,0.413206,-0.471763,-0.704225],[1,0,-5,0],[9E+09,9E+09,9E+09,9E+09,9E+09,9E+09]];
    CONST robtarget rB_v20_t98_c2 := [[-1181.81,1033.32,2627.22],[0.332817,0.413206,-0.471763,-0.704225],[0,0,-4,0],[9E+09,9E+09,9E+09,9E+09,9E+09,9E+09]];
    CONST jointtarget jA_v20_t98 := [[135.001,-11,-9.7,89.9993,14.7,-360],[9E+09,9E+09,9E+09,9E+09,9E+09,9E+09]];
    CONST jointtarget jB_v20_t98 := [[44.9994,-58.7,29.3,-90.0002,39.2,-360.001],[9E+09,9E+09,9E+09,9E+09,9E+09,9E+09]];
    CONST jointtarget jBseed_v20_t98 := [[135,-11,-9.7,90,14.7,-360],[9E+09,9E+09,9E+09,9E+09,9E+09,9E+09]];
    CONST num seedB_v20_t98 := 3251;

    CONST robtarget rA_v20_t99 := [[-1923.7,2060.11,1754.68],[0.480918,-0.753745,-0.39763,-0.2061],[1,-1,-2,0],[9E+09,9E+09,9E+09,9E+09,9E+09,9E+09]];
    CONST robtarget rB_v20_t99 := [[-1919.15,1974.28,1691.95],[0.524761,-0.726568,-0.363538,-0.254096],[1,-1,-2,0],[9E+09,9E+09,9E+09,9E+09,9E+09,9E+09]];
    CONST robtarget rB_v20_t99_c5 := [[-1919.15,1974.28,1691.95],[0.524761,-0.726568,-0.363538,-0.254096],[0,0,0,0],[9E+09,9E+09,9E+09,9E+09,9E+09,9E+09]];
    CONST jointtarget jA_v20_t99 := [[135.001,54,-65.4,-44.9991,54.8,-90.0002],[9E+09,9E+09,9E+09,9E+09,9E+09,9E+09]];
    CONST jointtarget jB_v20_t99 := [[44.9994,-58.7,29.3,-90.0002,39.2,-360.001],[9E+09,9E+09,9E+09,9E+09,9E+09,9E+09]];
    CONST jointtarget jBseed_v20_t99 := [[135,54,-65.4,-45,54.8,-90],[9E+09,9E+09,9E+09,9E+09,9E+09,9E+09]];
    CONST num seedB_v20_t99 := 17821;

    CONST robtarget rA_v20_t100 := [[2045.47,-1907.2,1677.43],[0.437618,0.416329,0.765746,0.220892],[-1,0,-5,0],[9E+09,9E+09,9E+09,9E+09,9E+09,9E+09]];
    CONST robtarget rB_v20_t100 := [[2085.59,-1975.84,1638.54],[0.392352,0.472261,0.762398,0.204397],[-1,0,-5,0],[9E+09,9E+09,9E+09,9E+09,9E+09,9E+09]];
    CONST robtarget rB_v20_t100_c2 := [[2085.59,-1975.84,1638.54],[0.392352,0.472261,0.762398,0.204397],[0,0,-4,0],[9E+09,9E+09,9E+09,9E+09,9E+09,9E+09]];
    CONST jointtarget jA_v20_t100 := [[-45.0001,49.8,-56.2,44.999,55.9,-360.001],[9E+09,9E+09,9E+09,9E+09,9E+09,9E+09]];
    CONST jointtarget jB_v20_t100 := [[44.9994,-58.7,29.3,-90.0002,39.2,-360.001],[9E+09,9E+09,9E+09,9E+09,9E+09,9E+09]];
    CONST jointtarget jBseed_v20_t100 := [[-45,49.8,-56.2,45,55.9,-360],[9E+09,9E+09,9E+09,9E+09,9E+09,9E+09]];
    CONST num seedB_v20_t100 := 14807;

    CONST robtarget rA_v20_t101 := [[-76.8521,-2218.78,2089.01],[0.713761,0.508911,0.0204297,-0.480767],[-2,2,2,0],[9E+09,9E+09,9E+09,9E+09,9E+09,9E+09]];
    CONST robtarget rB_v20_t101 := [[-90.741,-2153.91,2089.35],[0.675859,0.524003,0.0555649,-0.515313],[-2,2,2,0],[9E+09,9E+09,9E+09,9E+09,9E+09,9E+09]];
    CONST robtarget rB_v20_t101_c6 := [[-90.741,-2153.91,2089.35],[0.675859,0.524003,0.0555649,-0.515313],[0,4,0,0],[9E+09,9E+09,9E+09,9E+09,9E+09,9E+09]];
    CONST jointtarget jA_v20_t101 := [[-90.0001,12,-13.6,225.001,40.6,180],[9E+09,9E+09,9E+09,9E+09,9E+09,9E+09]];
    CONST jointtarget jB_v20_t101 := [[44.9994,-58.7,29.3,-90.0002,39.2,-360.001],[9E+09,9E+09,9E+09,9E+09,9E+09,9E+09]];
    CONST jointtarget jBseed_v20_t101 := [[-90,12,-13.6,225,40.6,180],[9E+09,9E+09,9E+09,9E+09,9E+09,9E+09]];
    CONST num seedB_v20_t101 := 13806;

    CONST robtarget rA_v20_t102 := [[-1174.59,-1207.9,1746.6],[0.466648,0.0469966,-0.697623,0.541621],[-2,-3,-4,0],[9E+09,9E+09,9E+09,9E+09,9E+09,9E+09]];
    CONST robtarget rB_v20_t102 := [[-1054.4,-1201.87,1728.82],[0.539185,0.0120691,-0.691608,0.48043],[-2,-3,-4,0],[9E+09,9E+09,9E+09,9E+09,9E+09,9E+09]];
    CONST robtarget rB_v20_t102_c1 := [[-1054.4,-1201.87,1728.82],[0.539185,0.0120691,-0.691608,0.48043],[0,-4,-4,0],[9E+09,9E+09,9E+09,9E+09,9E+09,9E+09]];
    CONST jointtarget jA_v20_t102 := [[-135,-18.8,25.7,-225.001,11.5,-270],[9E+09,9E+09,9E+09,9E+09,9E+09,9E+09]];
    CONST jointtarget jB_v20_t102 := [[44.9994,-58.7,29.3,-90.0002,39.2,-360.001],[9E+09,9E+09,9E+09,9E+09,9E+09,9E+09]];
    CONST jointtarget jBseed_v20_t102 := [[-135,-18.8,25.7,-225,11.5,-270],[9E+09,9E+09,9E+09,9E+09,9E+09,9E+09]];
    CONST num seedB_v20_t102 := 2851;

    CONST robtarget rA_v20_t103 := [[1469.05,1469.03,732.792],[0.428006,-0.796002,4.29286E-7,-0.428009],[0,1,0,0],[9E+09,9E+09,9E+09,9E+09,9E+09,9E+09]];
    CONST robtarget rB_v20_t103 := [[1533.28,1402.97,742.753],[0.411923,-0.832286,0.0400674,-0.368802],[0,1,0,0],[9E+09,9E+09,9E+09,9E+09,9E+09,9E+09]];
    CONST robtarget rB_v20_t103_c2 := [[1533.28,1402.97,742.753],[0.411923,-0.832286,0.0400674,-0.368802],[0,0,-4,0],[9E+09,9E+09,9E+09,9E+09,9E+09,9E+09]];
    CONST robtarget rB_v20_t103_c5 := [[1533.28,1402.97,742.753],[0.411923,-0.832286,0.0400674,-0.368802],[0,0,0,0],[9E+09,9E+09,9E+09,9E+09,9E+09,9E+09]];
    CONST jointtarget jA_v20_t103 := [[44.9997,18.8,26.2,180,29.5,44.9999],[9E+09,9E+09,9E+09,9E+09,9E+09,9E+09]];
    CONST jointtarget jB_v20_t103 := [[44.9994,-58.7,29.3,-90.0002,39.2,-360.001],[9E+09,9E+09,9E+09,9E+09,9E+09,9E+09]];
    CONST jointtarget jBseed_v20_t103 := [[45,18.8,26.2,180,29.5,45],[9E+09,9E+09,9E+09,9E+09,9E+09,9E+09]];
    CONST num seedB_v20_t103 := 10355;

    CONST robtarget rA_v20_t104 := [[-1547.49,1485.42,1425.34],[0.0823732,-0.833881,0.259519,0.480112],[1,0,3,0],[9E+09,9E+09,9E+09,9E+09,9E+09,9E+09]];
    CONST robtarget rB_v20_t104 := [[-1555.55,1467.19,1469.64],[0.1228,-0.827789,0.197425,0.510596],[1,0,3,0],[9E+09,9E+09,9E+09,9E+09,9E+09,9E+09]];
    CONST robtarget rB_v20_t104_c8 := [[-1555.55,1467.19,1469.64],[0.1228,-0.827789,0.197425,0.510596],[0,0,4,0],[9E+09,9E+09,9E+09,9E+09,9E+09,9E+09]];
    CONST jointtarget jA_v20_t104 := [[135.001,7.8,9.4,44.9998,21.8,315.001],[9E+09,9E+09,9E+09,9E+09,9E+09,9E+09]];
    CONST jointtarget jB_v20_t104 := [[44.9994,-58.7,29.3,-90.0002,39.2,-360.001],[9E+09,9E+09,9E+09,9E+09,9E+09,9E+09]];
    CONST jointtarget jBseed_v20_t104 := [[135,7.8,9.4,45,21.8,315],[9E+09,9E+09,9E+09,9E+09,9E+09,9E+09]];
    CONST num seedB_v20_t104 := 8562;

    CONST robtarget rA_v20_t105 := [[-90.7233,-83.5297,3205.12],[0.900563,-0.206253,-0.231904,0.304411],[-1,2,-2,0],[9E+09,9E+09,9E+09,9E+09,9E+09,9E+09]];
    CONST robtarget rB_v20_t105 := [[-110.105,-56.3223,3265.61],[0.874359,-0.22406,-0.220971,0.369411],[-1,2,-2,0],[9E+09,9E+09,9E+09,9E+09,9E+09,9E+09]];
    CONST robtarget rB_v20_t105_c6 := [[-110.105,-56.3223,3265.61],[0.874359,-0.22406,-0.220971,0.369411],[0,4,0,0],[9E+09,9E+09,9E+09,9E+09,9E+09,9E+09]];
    CONST jointtarget jA_v20_t105 := [[-89.9995,-35.8,-29.8,225,50.2,-90.0009],[9E+09,9E+09,9E+09,9E+09,9E+09,9E+09]];
    CONST jointtarget jB_v20_t105 := [[44.9994,-58.7,29.3,-90.0002,39.2,-360.001],[9E+09,9E+09,9E+09,9E+09,9E+09,9E+09]];
    CONST jointtarget jBseed_v20_t105 := [[-90,-35.8,-29.8,225,50.2,-90],[9E+09,9E+09,9E+09,9E+09,9E+09,9E+09]];
    CONST num seedB_v20_t105 := 11833;

    CONST robtarget rA_v20_t106 := [[2022.52,-64.6798,2131.95],[0.488894,-0.16082,0.783921,-0.347257],[-1,-1,3,0],[9E+09,9E+09,9E+09,9E+09,9E+09,9E+09]];
    CONST robtarget rB_v20_t106 := [[2109.69,-135.651,2177.61],[0.52262,-0.113825,0.7959,-0.283646],[-1,-1,3,0],[9E+09,9E+09,9E+09,9E+09,9E+09,9E+09]];
    CONST robtarget rB_v20_t106_c8 := [[2109.69,-135.651,2177.61],[0.52262,-0.113825,0.7959,-0.283646],[0,0,4,0],[9E+09,9E+09,9E+09,9E+09,9E+09,9E+09]];
    CONST jointtarget jA_v20_t106 := [[-0.000558583,2.3,-9.4,-45.0001,33.2,359.999],[9E+09,9E+09,9E+09,9E+09,9E+09,9E+09]];
    CONST jointtarget jB_v20_t106 := [[44.9994,-58.7,29.3,-90.0002,39.2,-360.001],[9E+09,9E+09,9E+09,9E+09,9E+09,9E+09]];
    CONST jointtarget jBseed_v20_t106 := [[0,2.3,-9.4,-45,33.2,360],[9E+09,9E+09,9E+09,9E+09,9E+09,9E+09]];
    CONST num seedB_v20_t106 := 25059;

    CONST robtarget rA_v20_t107 := [[-42.3685,1229.85,1644.67],[0.430465,-0.560987,0.433389,0.558719],[0,-4,-2,0],[9E+09,9E+09,9E+09,9E+09,9E+09,9E+09]];
    CONST robtarget rB_v20_t107 := [[-116.562,1186.37,1657],[0.518002,-0.500478,0.416134,0.555003],[0,-4,-2,0],[9E+09,9E+09,9E+09,9E+09,9E+09,9E+09]];
    CONST robtarget rB_v20_t107_c1 := [[-116.562,1186.37,1657],[0.518002,-0.500478,0.416134,0.555003],[0,-4,-4,0],[9E+09,9E+09,9E+09,9E+09,9E+09,9E+09]];
    CONST jointtarget jA_v20_t107 := [[89.9996,-45.6,45.9,-270,14.7,-90.0005],[9E+09,9E+09,9E+09,9E+09,9E+09,9E+09]];
    CONST jointtarget jB_v20_t107 := [[44.9994,-58.7,29.3,-90.0002,39.2,-360.001],[9E+09,9E+09,9E+09,9E+09,9E+09,9E+09]];
    CONST jointtarget jBseed_v20_t107 := [[90,-45.6,45.9,-270,14.7,-90],[9E+09,9E+09,9E+09,9E+09,9E+09,9E+09]];
    CONST num seedB_v20_t107 := 28946;

    CONST robtarget rA_v20_t109 := [[1245.62,1367.34,2986.03],[0.950217,-0.275279,-0.0843582,0.119129],[0,1,1,0],[9E+09,9E+09,9E+09,9E+09,9E+09,9E+09]];
    CONST robtarget rB_v20_t109 := [[1259.69,1323.05,3004.38],[0.940753,-0.287076,-0.0318827,0.177635],[0,1,1,0],[9E+09,9E+09,9E+09,9E+09,9E+09,9E+09]];
    CONST robtarget rB_v20_t109_c5 := [[1259.69,1323.05,3004.38],[0.940753,-0.287076,-0.0318827,0.177635],[0,0,0,0],[9E+09,9E+09,9E+09,9E+09,9E+09,9E+09]];
    CONST jointtarget jA_v20_t109 := [[44.9998,22.8,-62.6,135.001,46.8,180],[9E+09,9E+09,9E+09,9E+09,9E+09,9E+09]];
    CONST jointtarget jB_v20_t109 := [[44.9994,-58.7,29.3,-90.0002,39.2,-360.001],[9E+09,9E+09,9E+09,9E+09,9E+09,9E+09]];
    CONST jointtarget jBseed_v20_t109 := [[45,22.8,-62.6,135,46.8,180],[9E+09,9E+09,9E+09,9E+09,9E+09,9E+09]];
    CONST num seedB_v20_t109 := 13077;

    CONST robtarget rA_v20_t110 := [[1577.74,80.7038,2206.79],[0.561424,-0.202276,0.785711,0.162928],[0,0,-1,0],[9E+09,9E+09,9E+09,9E+09,9E+09,9E+09]];
    CONST robtarget rB_v20_t110 := [[1570.3,21.1613,2163.96],[0.492643,-0.175313,0.825578,0.212106],[0,0,-1,0],[9E+09,9E+09,9E+09,9E+09,9E+09,9E+09]];
    CONST robtarget rB_v20_t110_c5 := [[1570.3,21.1613,2163.96],[0.492643,-0.175313,0.825578,0.212106],[0,0,0,0],[9E+09,9E+09,9E+09,9E+09,9E+09,9E+09]];
    CONST jointtarget jA_v20_t110 := [[0.000683653,-18.1,5.8,44.9995,43.1,-44.9992],[9E+09,9E+09,9E+09,9E+09,9E+09,9E+09]];
    CONST jointtarget jB_v20_t110 := [[44.9994,-58.7,29.3,-90.0002,39.2,-360.001],[9E+09,9E+09,9E+09,9E+09,9E+09,9E+09]];
    CONST jointtarget jBseed_v20_t110 := [[0,-18.1,5.8,45,43.1,-45],[9E+09,9E+09,9E+09,9E+09,9E+09,9E+09]];
    CONST num seedB_v20_t110 := 20798;

    CONST robtarget rA_v20_t111 := [[334.264,76.2184,3131.58],[0.768179,-0.042989,0.51328,0.380259],[-1,0,3,0],[9E+09,9E+09,9E+09,9E+09,9E+09,9E+09]];
    CONST robtarget rB_v20_t111 := [[388.374,43.6512,3148.43],[0.805026,-0.0361462,0.457829,0.375524],[-1,0,3,0],[9E+09,9E+09,9E+09,9E+09,9E+09,9E+09]];
    CONST robtarget rB_v20_t111_c8 := [[388.374,43.6512,3148.43],[0.805026,-0.0361462,0.457829,0.375524],[0,0,4,0],[9E+09,9E+09,9E+09,9E+09,9E+09,9E+09]];
    CONST jointtarget jA_v20_t111 := [[-0.000308544,-35.1,-27.6,45.0001,40.2,360],[9E+09,9E+09,9E+09,9E+09,9E+09,9E+09]];
    CONST jointtarget jB_v20_t111 := [[44.9994,-58.7,29.3,-90.0002,39.2,-360.001],[9E+09,9E+09,9E+09,9E+09,9E+09,9E+09]];
    CONST jointtarget jBseed_v20_t111 := [[0,-35.1,-27.6,45,40.2,360],[9E+09,9E+09,9E+09,9E+09,9E+09,9E+09]];
    CONST num seedB_v20_t111 := 7831;

    CONST robtarget rA_v20_t112 := [[-1644.58,-1550.93,1566.25],[0.0232884,0.854166,0.211224,-0.474598],[-2,-1,0,0],[9E+09,9E+09,9E+09,9E+09,9E+09,9E+09]];
    CONST robtarget rB_v20_t112 := [[-1530.11,-1522.35,1553.23],[0.0717775,0.847546,0.241972,-0.466866],[-2,-1,0,0],[9E+09,9E+09,9E+09,9E+09,9E+09,9E+09]];
    CONST robtarget rB_v20_t112_c5 := [[-1530.11,-1522.35,1553.23],[0.0717775,0.847546,0.241972,-0.466866],[0,0,0,0],[9E+09,9E+09,9E+09,9E+09,9E+09,9E+09]];
    CONST jointtarget jA_v20_t112 := [[-135,13.4,-2.3,-45.001,34.1,44.9993],[9E+09,9E+09,9E+09,9E+09,9E+09,9E+09]];
    CONST jointtarget jB_v20_t112 := [[44.9994,-58.7,29.3,-90.0002,39.2,-360.001],[9E+09,9E+09,9E+09,9E+09,9E+09,9E+09]];
    CONST jointtarget jBseed_v20_t112 := [[-135,13.4,-2.3,-45,34.1,45],[9E+09,9E+09,9E+09,9E+09,9E+09,9E+09]];
    CONST num seedB_v20_t112 := 30210;

    CONST robtarget rA_v20_t113 := [[1671.45,1671.42,2147.22],[0.567673,-0.596225,4.32688E-7,-0.567683],[0,-3,-4,0],[9E+09,9E+09,9E+09,9E+09,9E+09,9E+09]];
    CONST robtarget rB_v20_t113 := [[1602.95,1659.55,2191.52],[0.565956,-0.563904,0.0283902,-0.60075],[0,-3,-4,0],[9E+09,9E+09,9E+09,9E+09,9E+09,9E+09]];
    CONST robtarget rB_v20_t113_c1 := [[1602.95,1659.55,2191.52],[0.565956,-0.563904,0.0283902,-0.60075],[0,-4,-4,0],[9E+09,9E+09,9E+09,9E+09,9E+09,9E+09]];
    CONST jointtarget jA_v20_t113 := [[44.9994,19.2,-25.6,-180,10.4,-315],[9E+09,9E+09,9E+09,9E+09,9E+09,9E+09]];
    CONST jointtarget jB_v20_t113 := [[44.9994,-58.7,29.3,-90.0002,39.2,-360.001],[9E+09,9E+09,9E+09,9E+09,9E+09,9E+09]];
    CONST jointtarget jBseed_v20_t113 := [[45,19.2,-25.6,-180,10.4,-315],[9E+09,9E+09,9E+09,9E+09,9E+09,9E+09]];
    CONST num seedB_v20_t113 := 11870;

    CONST robtarget rA_v20_t114 := [[-0.00502908,-2150.79,1.27949],[2.98185E-6,7.5229E-6,-0.938794,0.344479],[-2,-3,0,0],[9E+09,9E+09,9E+09,9E+09,9E+09,9E+09]];
    CONST robtarget rB_v20_t114 := [[-44.1494,-2166.86,25.2112],[0.00958077,-0.0931687,0.94665,-0.308354],[-2,-3,0,0],[9E+09,9E+09,9E+09,9E+09,9E+09,9E+09]];
    CONST robtarget rB_v20_t114_c4 := [[-44.1494,-2166.86,25.2112],[0.00958077,-0.0931687,0.94665,-0.308354],[0,-4,0,0],[9E+09,9E+09,9E+09,9E+09,9E+09,9E+09]];
    CONST robtarget rB_v20_t114_c5 := [[-44.1494,-2166.86,25.2112],[0.00958077,-0.0931687,0.94665,-0.308354],[0,0,0,0],[9E+09,9E+09,9E+09,9E+09,9E+09,9E+09]];
    CONST jointtarget jA_v20_t114 := [[-90.0001,48.4,14.4,-180,13.1,89.9993],[9E+09,9E+09,9E+09,9E+09,9E+09,9E+09]];
    CONST jointtarget jB_v20_t114 := [[44.9994,-58.7,29.3,-90.0002,39.2,-360.001],[9E+09,9E+09,9E+09,9E+09,9E+09,9E+09]];
    CONST jointtarget jBseed_v20_t114 := [[-90,48.4,14.4,-180,13.1,90],[9E+09,9E+09,9E+09,9E+09,9E+09,9E+09]];
    CONST num seedB_v20_t114 := 31163;

    CONST robtarget rA_v20_t115 := [[2020.89,2011.84,802.327],[0.190613,-0.78299,-0.313177,-0.502507],[0,2,-2,0],[9E+09,9E+09,9E+09,9E+09,9E+09,9E+09]];
    CONST robtarget rB_v20_t115 := [[2022.24,2085.68,726.679],[0.122165,-0.800281,-0.278482,-0.516793],[0,2,-2,0],[9E+09,9E+09,9E+09,9E+09,9E+09,9E+09]];
    CONST robtarget rB_v20_t115_c6 := [[2022.24,2085.68,726.679],[0.122165,-0.800281,-0.278482,-0.516793],[0,4,0,0],[9E+09,9E+09,9E+09,9E+09,9E+09,9E+09]];
    CONST jointtarget jA_v20_t115 := [[45.0004,52.9,-27.9,269.999,2.2,-90.0008],[9E+09,9E+09,9E+09,9E+09,9E+09,9E+09]];
    CONST jointtarget jB_v20_t115 := [[44.9994,-58.7,29.3,-90.0002,39.2,-360.001],[9E+09,9E+09,9E+09,9E+09,9E+09,9E+09]];
    CONST jointtarget jBseed_v20_t115 := [[45,52.9,-27.9,270,2.2,-90],[9E+09,9E+09,9E+09,9E+09,9E+09,9E+09]];
    CONST num seedB_v20_t115 := 28940;

    CONST robtarget rA_v20_t116 := [[-1568.29,-1744.89,1497.44],[0.0870797,0.0454774,0.763365,-0.638453],[-2,1,-3,0],[9E+09,9E+09,9E+09,9E+09,9E+09,9E+09]];
    CONST robtarget rB_v20_t116 := [[-1561.04,-1740.57,1510.11],[0.0724004,0.14239,0.737994,-0.655628],[-2,1,-3,0],[9E+09,9E+09,9E+09,9E+09,9E+09,9E+09]];
    CONST robtarget rB_v20_t116_c1 := [[-1561.04,-1740.57,1510.11],[0.0724004,0.14239,0.737994,-0.655628],[0,-4,-4,0],[9E+09,9E+09,9E+09,9E+09,9E+09,9E+09]];
    CONST robtarget rB_v20_t116_c2 := [[-1561.04,-1740.57,1510.11],[0.0724004,0.14239,0.737994,-0.655628],[0,0,-4,0],[9E+09,9E+09,9E+09,9E+09,9E+09,9E+09]];
    CONST jointtarget jA_v20_t116 := [[-135,19.2,-4.4,90.0007,48.4,-180.001],[9E+09,9E+09,9E+09,9E+09,9E+09,9E+09]];
    CONST jointtarget jB_v20_t116 := [[44.9994,-58.7,29.3,-90.0002,39.2,-360.001],[9E+09,9E+09,9E+09,9E+09,9E+09,9E+09]];
    CONST jointtarget jBseed_v20_t116 := [[-135,19.2,-4.4,90,48.4,-180],[9E+09,9E+09,9E+09,9E+09,9E+09,9E+09]];
    CONST num seedB_v20_t116 := 6791;

    CONST robtarget rA_v20_t117 := [[-60.4148,2112.48,52.5841],[0.178253,0.0454405,-0.95248,-0.24278],[1,-4,-4,0],[9E+09,9E+09,9E+09,9E+09,9E+09,9E+09]];
    CONST robtarget rB_v20_t117 := [[8.06042,2073.24,55.1007],[0.157937,0.0928747,-0.959923,-0.21208],[1,-4,-4,0],[9E+09,9E+09,9E+09,9E+09,9E+09,9E+09]];
    CONST robtarget rB_v20_t117_c1 := [[8.06042,2073.24,55.1007],[0.157937,0.0928747,-0.959923,-0.21208],[0,-4,-4,0],[9E+09,9E+09,9E+09,9E+09,9E+09,9E+09]];
    CONST jointtarget jA_v20_t117 := [[90.0006,45.7,15.7,-270.001,21.2,-359.999],[9E+09,9E+09,9E+09,9E+09,9E+09,9E+09]];
    CONST jointtarget jB_v20_t117 := [[44.9994,-58.7,29.3,-90.0002,39.2,-360.001],[9E+09,9E+09,9E+09,9E+09,9E+09,9E+09]];
    CONST jointtarget jBseed_v20_t117 := [[90,45.7,15.7,-270,21.2,-360],[9E+09,9E+09,9E+09,9E+09,9E+09,9E+09]];
    CONST num seedB_v20_t117 := 22567;

    CONST robtarget rA_v20_t118 := [[-104.23,2803.15,663.541],[0.136129,-0.693886,0.457343,0.539285],[1,-4,-1,0],[9E+09,9E+09,9E+09,9E+09,9E+09,9E+09]];
    CONST robtarget rB_v20_t118 := [[-214.228,2759.09,591.047],[0.0911861,-0.65524,0.460802,0.591614],[1,-4,-1,0],[9E+09,9E+09,9E+09,9E+09,9E+09,9E+09]];
    CONST robtarget rB_v20_t118_c4 := [[-214.228,2759.09,591.047],[0.0911861,-0.65524,0.460802,0.591614],[0,-4,0,0],[9E+09,9E+09,9E+09,9E+09,9E+09,9E+09]];
    CONST jointtarget jA_v20_t118 := [[90.0009,55.3,-26.1,-270.001,38.6,-89.9997],[9E+09,9E+09,9E+09,9E+09,9E+09,9E+09]];
    CONST jointtarget jB_v20_t118 := [[44.9994,-58.7,29.3,-90.0002,39.2,-360.001],[9E+09,9E+09,9E+09,9E+09,9E+09,9E+09]];
    CONST jointtarget jBseed_v20_t118 := [[90,55.3,-26.1,-270,38.6,-90],[9E+09,9E+09,9E+09,9E+09,9E+09,9E+09]];
    CONST num seedB_v20_t118 := 25276;

    CONST robtarget rA_v20_t119 := [[2699.69,41.525,2047.24],[0.394916,-0.52993,0.11445,-0.741699],[-1,1,-3,0],[9E+09,9E+09,9E+09,9E+09,9E+09,9E+09]];
    CONST robtarget rB_v20_t119 := [[2662.65,73.8312,2128.79],[0.428133,-0.476924,0.0573235,-0.76548],[-1,1,-3,0],[9E+09,9E+09,9E+09,9E+09,9E+09,9E+09]];
    CONST robtarget rB_v20_t119_c2 := [[2662.65,73.8312,2128.79],[0.428133,-0.476924,0.0573235,-0.76548],[0,0,-4,0],[9E+09,9E+09,9E+09,9E+09,9E+09,9E+09]];
    CONST jointtarget jA_v20_t119 := [[-0.000482366,41.8,-52.1,135,20.6,-269.999],[9E+09,9E+09,9E+09,9E+09,9E+09,9E+09]];
    CONST jointtarget jB_v20_t119 := [[44.9994,-58.7,29.3,-90.0002,39.2,-360.001],[9E+09,9E+09,9E+09,9E+09,9E+09,9E+09]];
    CONST jointtarget jBseed_v20_t119 := [[0,41.8,-52.1,135,20.6,-270],[9E+09,9E+09,9E+09,9E+09,9E+09,9E+09]];
    CONST num seedB_v20_t119 := 13315;

    CONST robtarget rA_v20_t120 := [[1601.93,-1601.88,2270.55],[0.350532,0.370614,-0.153511,0.84629],[-1,-3,0,0],[9E+09,9E+09,9E+09,9E+09,9E+09,9E+09]];
    CONST robtarget rB_v20_t120 := [[1691.03,-1555.08,2267.87],[0.371834,0.334011,-0.0415908,0.865128],[-1,-3,0,0],[9E+09,9E+09,9E+09,9E+09,9E+09,9E+09]];
    CONST robtarget rB_v20_t120_c4 := [[1691.03,-1555.08,2267.87],[0.371834,0.334011,-0.0415908,0.865128],[0,-4,0,0],[9E+09,9E+09,9E+09,9E+09,9E+09,9E+09]];
    CONST robtarget rB_v20_t120_c5 := [[1691.03,-1555.08,2267.87],[0.371834,0.334011,-0.0415908,0.865128],[0,0,0,0],[9E+09,9E+09,9E+09,9E+09,9E+09,9E+09]];
    CONST jointtarget jA_v20_t120 := [[-44.9991,16.5,-24.5,-180,34.7,0.000703174],[9E+09,9E+09,9E+09,9E+09,9E+09,9E+09]];
    CONST jointtarget jB_v20_t120 := [[44.9994,-58.7,29.3,-90.0002,39.2,-360.001],[9E+09,9E+09,9E+09,9E+09,9E+09,9E+09]];
    CONST jointtarget jBseed_v20_t120 := [[-45,16.5,-24.5,-180,34.7,0],[9E+09,9E+09,9E+09,9E+09,9E+09,9E+09]];
    CONST num seedB_v20_t120 := 30820;

    CONST robtarget rA_v20_t121 := [[2320.78,-0.0136512,658.271],[0.434363,0.557973,0.557961,0.434367],[-1,2,3,0],[9E+09,9E+09,9E+09,9E+09,9E+09,9E+09]];
    CONST robtarget rB_v20_t121 := [[2235.44,-9.77427,696.794],[0.440625,0.583121,0.595689,0.333127],[-1,2,3,0],[9E+09,9E+09,9E+09,9E+09,9E+09,9E+09]];
    CONST robtarget rB_v20_t121_c8 := [[2235.44,-9.77427,696.794],[0.440625,0.583121,0.595689,0.333127],[0,0,4,0],[9E+09,9E+09,9E+09,9E+09,9E+09,9E+09]];
    CONST jointtarget jA_v20_t121 := [[-0.000334904,31.4,12.4,180,29.6,270.001],[9E+09,9E+09,9E+09,9E+09,9E+09,9E+09]];
    CONST jointtarget jB_v20_t121 := [[44.9994,-58.7,29.3,-90.0002,39.2,-360.001],[9E+09,9E+09,9E+09,9E+09,9E+09,9E+09]];
    CONST jointtarget jBseed_v20_t121 := [[0,31.4,12.4,180,29.6,270],[9E+09,9E+09,9E+09,9E+09,9E+09,9E+09]];
    CONST num seedB_v20_t121 := 10657;

    CONST robtarget rA_v20_t122 := [[-1697.04,1736.8,1010.13],[0.43935,-0.368192,-0.776771,-0.260832],[1,-2,-1,0],[9E+09,9E+09,9E+09,9E+09,9E+09,9E+09]];
    CONST robtarget rB_v20_t122 := [[-1726.41,1725.64,1039.68],[0.369771,-0.327761,-0.812321,-0.309801],[1,-2,-1,0],[9E+09,9E+09,9E+09,9E+09,9E+09,9E+09]];
    CONST robtarget rB_v20_t122_c5 := [[-1726.41,1725.64,1039.68],[0.369771,-0.327761,-0.812321,-0.309801],[0,0,0,0],[9E+09,9E+09,9E+09,9E+09,9E+09,9E+09]];
    CONST robtarget rB_v20_t122_c8 := [[-1726.41,1725.64,1039.68],[0.369771,-0.327761,-0.812321,-0.309801],[0,0,4,0],[9E+09,9E+09,9E+09,9E+09,9E+09,9E+09]];
    CONST jointtarget jA_v20_t122 := [[135.001,27.3,1.7,-90.0005,9.7,-89.9993],[9E+09,9E+09,9E+09,9E+09,9E+09,9E+09]];
    CONST jointtarget jB_v20_t122 := [[44.9994,-58.7,29.3,-90.0002,39.2,-360.001],[9E+09,9E+09,9E+09,9E+09,9E+09,9E+09]];
    CONST jointtarget jBseed_v20_t122 := [[135,27.3,1.7,-90,9.7,-90],[9E+09,9E+09,9E+09,9E+09,9E+09,9E+09]];
    CONST num seedB_v20_t122 := 14948;

    CONST robtarget rA_v20_t123 := [[-1689.04,-1688.99,704.1],[0.0525963,-0.379068,-0.915105,0.126983],[-2,0,-1,0],[9E+09,9E+09,9E+09,9E+09,9E+09,9E+09]];
    CONST robtarget rB_v20_t123 := [[-1606.07,-1662.92,683.904],[0.105677,-0.424374,-0.880144,0.184622],[-2,0,-1,0],[9E+09,9E+09,9E+09,9E+09,9E+09,9E+09]];
    CONST robtarget rB_v20_t123_c5 := [[-1606.07,-1662.92,683.904],[0.105677,-0.424374,-0.880144,0.184622],[0,0,0,0],[9E+09,9E+09,9E+09,9E+09,9E+09,9E+09]];
    CONST jointtarget jA_v20_t123 := [[-135.001,34.9,0.1,0.00023244,39.2,-89.999],[9E+09,9E+09,9E+09,9E+09,9E+09,9E+09]];
    CONST jointtarget jB_v20_t123 := [[44.9994,-58.7,29.3,-90.0002,39.2,-360.001],[9E+09,9E+09,9E+09,9E+09,9E+09,9E+09]];
    CONST jointtarget jBseed_v20_t123 := [[-135,34.9,0.1,0,39.2,-90],[9E+09,9E+09,9E+09,9E+09,9E+09,9E+09]];
    CONST num seedB_v20_t123 := 26807;

    CONST robtarget rA_v20_t124 := [[1767.67,1810.35,1059.06],[0.521387,-0.349187,0.718497,0.299976],[0,-3,2,0],[9E+09,9E+09,9E+09,9E+09,9E+09,9E+09]];
    CONST robtarget rB_v20_t124 := [[1754.62,1771.35,1025.94],[0.448066,-0.426462,0.724636,0.30376],[0,-3,2,0],[9E+09,9E+09,9E+09,9E+09,9E+09,9E+09]];
    CONST robtarget rB_v20_t124_c7 := [[1754.62,1771.35,1025.94],[0.448066,-0.426462,0.724636,0.30376],[0,-4,4,0],[9E+09,9E+09,9E+09,9E+09,9E+09,9E+09]];
    CONST jointtarget jA_v20_t124 := [[45.0004,31.3,-4.4,-225,14.8,225],[9E+09,9E+09,9E+09,9E+09,9E+09,9E+09]];
    CONST jointtarget jB_v20_t124 := [[44.9994,-58.7,29.3,-90.0002,39.2,-360.001],[9E+09,9E+09,9E+09,9E+09,9E+09,9E+09]];
    CONST jointtarget jBseed_v20_t124 := [[45,31.3,-4.4,-225,14.8,225],[9E+09,9E+09,9E+09,9E+09,9E+09,9E+09]];
    CONST num seedB_v20_t124 := 8330;

